(*~
        <docu>
            <summary>
                Clears the message content.
                <remarks>
                    <note type="important">
                        This method is exposed for Rpc calls, for testing purposes. Rpc calls of this method must not be used in production code
                    </note>
                </remarks>
            </summary>
        </docu>
~*)
{attribute 'TcRpcEnable'}
METHOD Clear
_mime.TimeStamp := DT#1970-01-01-00:00;
_mime.Text := '';
_mime.Identity := 0;
_mime.Category := eMessageCategory.All;
_mime.Cycle := 0;
_mime.PerCycleCount := 0;
_mime.Pinned := FALSE;
END_METHOD

METHOD PROTECTED Compose : TcoMessage
VAR_INPUT
    Text : STRING(TcoMessengerEnv.MAX_MESSAGE_TEXT_LENGHT);
    Category : eMessageCategory;
END_VAR
IF (_Parent <> 0 AND_THEN _Parent.Context <> 0 AND_THEN _Parent.Context.RealTimeClock <> 0) THEN
    Compose.TimeStamp := _Parent.Context.RealTimeClock.NowLocal();
    Compose.Text := Text;
    Compose.Identity := _Parent.Identity;
    Compose.Category := Category;
    Compose.Cycle := _Parent.Context.StartCycleCount;
    Compose.MessageDigest := Digest(Text, THIS^._Parent.Context.Environment.Messaging.MessageDigestMethod);
END_IF;
END_METHOD

(*~
        <docu>
            <summary>
                Adds message of 'critical' category to the message queue.
                Use this category when a critical error occured, that is not recoverable by the means of software (reset/restore) and a detailed inspection is required.
            </summary>
        </docu>
~*)
METHOD PUBLIC Critical : ITcoMessageProperties
VAR_INPUT
    (*~
        <docu>
            <summary>
                Arbitrary message string.
            </summary>
        </docu>
    ~*)
    Message : STRING(TcoMessengerEnv.MAX_MESSAGE_TEXT_LENGHT);
END_VAR
Critical := THIS^.Post(Message, eMessageCategory.Critical);
END_METHOD

(*~
        <docu>
            <summary>
                Adds message of 'debug' category to the message queue.
                Use when you need to report debug information for you as programmer.
            </summary>
        </docu>
~*)
METHOD PUBLIC Debug : ITcoMessageProperties
VAR_INPUT
    (*~
        <docu>
            <summary>
                Arbitrary message string.
            </summary>
        </docu>
    ~*)
    Message : STRING(TcoMessengerEnv.MAX_MESSAGE_TEXT_LENGHT);
END_VAR
Debug := THIS^.Post(Message, eMessageCategory.Debug);
END_METHOD

METHOD Digest : DWORD
VAR_INPUT
    Text : Tc2_System.T_MaxString;
    inDigestType : eMessageDigestMethod;
END_VAR
CASE inDigestType OF
    eMessageDigestMethod.CRC8:
        Digest := TcoCRC_8(Text);
    eMessageDigestMethod.CRC16:
        Digest := TcoCRC_16(Text);
    eMessageDigestMethod.CRC32:
        Digest := TcoCRC_32(Text);
ELSE
    Digest := 0;
END_CASE
END_METHOD

(*~
        <docu>
            <summary>
                Adds message of 'error' category to the message queue.
                Use this categoty when there is a failure that cannot be immediately recovered and an intervention is needed. This is typically a situation when a device fails
                to deliver expected result.
                Do not use this category to report information about failed process like measurement or detection.
            </summary>
        </docu>
~*)
METHOD PUBLIC Error : ITcoMessageProperties
VAR_INPUT
    (*~
        <docu>
            <summary>
                Arbitrary message string.
            </summary>
        </docu>
    ~*)
    Message : STRING(TcoMessengerEnv.MAX_MESSAGE_TEXT_LENGHT);
END_VAR
Error := THIS^.Post(Message, eMessageCategory.Error);
END_METHOD

{attribute 'hide'}
METHOD FB_init : BOOL
VAR_INPUT
    bInitRetains : BOOL; // if TRUE, the retain variables are initialized (warm start / cold start)
    bInCopyCode : BOOL; // if TRUE, the instance afterwards gets moved into the copy code (online change)
    ParentObject : ITcoObject;
END_VAR
_Parent := ParentObject;
_contextIdentity := ParentObject.Identity;
END_METHOD

(*~
        <docu>
            <summary>
                Adds message of 'information' category to the message queue.
                Use when you want to deliver information to the user, that has only informative character and does not adversely affect a process.
            </summary>
        </docu>
~*)
METHOD PUBLIC Info : ITcoMessageProperties
VAR_INPUT
    (*~
        <docu>
            <summary>
                Arbitrary message string.
            </summary>
        </docu>
    ~*)
    Message : STRING(TcoMessengerEnv.MAX_MESSAGE_TEXT_LENGHT);
END_VAR
Info := THIS^.Post(Message, eMessageCategory.Info);
END_METHOD

METHOD PRIVATE LogMessage
VAR_IN_OUT
    inMessage : TcoMessage;
END_VAR
VAR
    _index : INT;
    _freeIndex : INT;
END_VAR
CASE _Parent.Context.Environment.Messaging.MessengerLoggingMethod OF
    eMessengerLogMethod.OnEventRisen:
        IF (_Parent.Context.Environment.Messaging.MessageDigestMethod = eMessageDigestMethod.NONE) THEN
            inMessage.MessageDigest := Digest(inMessage.Text, eMessageDigestMethod.CRC32);
        END_IF

        _freeIndex := 0;

        FOR _index := 0 TO MDS_MAX_INDEX DO
            IF (_mds[_index].Cycle = inMessage.Cycle - 1 OR _mds[_index].Cycle = inMessage.Cycle) AND_THEN
                (_mds[_index].Digest = inMessage.MessageDigest) AND_THEN
                (_mds[_index].Category = inMessage.Category) THEN
                _mds[_index].Cycle := inMessage.Cycle;
                RETURN;
            END_IF

            IF ((_mds[_index].Cycle <> inMessage.Cycle - 1) AND (_mds[_index].Cycle <> inMessage.Cycle)) THEN
                _freeIndex := _index;
            END_IF
        END_FOR

        IF (_freeIndex <= THIS^.MDS_MAX_INDEX) THEN
            _mds[_freeIndex].Digest := inMessage.MessageDigest;
            _mds[_freeIndex].Cycle := inMessage.Cycle;
            _mds[_freeIndex].Category := inMessage.Category;
            _Parent.Context.Logger.PushMessage(inMessage);
        END_IF;
    eMessengerLogMethod.Continuous:
        _Parent.Context.Logger.PushMessage(inMessage);
END_CASE
END_METHOD

(*~
        <docu>
            <summary>
                Adds message of 'notification' category to the message queue.
                Use this category when you want to report a notification that may be of interest to the user, but does not adveresly affect a process.
            </summary>
        </docu>
~*)
METHOD Notify : ITcoMessageProperties
VAR_INPUT
    (*~
        <docu>
            <summary>
                Arbitrary message string.
            </summary>
        </docu>
    ~*)
    Message : STRING(TcoMessengerEnv.MAX_MESSAGE_TEXT_LENGHT);
END_VAR
Notify := THIS^.Post(Message, eMessageCategory.Notification);
END_METHOD

METHOD OnCondition : ITcoMessages
VAR_INPUT
    inCondition : BOOL;
END_VAR
IF (inCondition) THEN
    _condition := eMessageCondition.Active;
ELSE
    _condition := eMessageCondition.Inactive;
END_IF

OnCondition := THIS^;
END_METHOD

(*~
    <docu>
        <summary>
            Pins this message that no other message will override it.
            The messenger won't accept new messages until acknowledged in diagnostics view by user, unipenned by `Unpin()` methods or cleared by `Clear()` method
            of this messenger.
        </summary>
        <note type="important">
            Pinned messages do no accept incomming messages on the same messenger. The incomming messages will be though the context logger when active.
        </note>
    </docu>
~*)
//~
{attribute 'hide'}
{attribute 'obsolete' := 'This method must be called exclusively over ITcoMessageProperties interface'}
//~
METHOD Pin : ITcoMessageProperties
IF (_Parent <> 0 AND_THEN _Parent.Context <> 0) THEN
    IF (_pinnable AND_THEN _mime.Cycle = _Parent.Context.StartCycleCount) THEN
        _mime.Pinned := TRUE;
    END_IF;
END_IF;

Pin := THIS^;
END_METHOD

(*~
    <docu>
        <summary>
            Gets `true` when this messanger is pinned (awaiting acknowledgement in diagnostics view).
        </summary>
    </docu>
~*)
PROPERTY Pinned : BOOL
GET
Pinned := _mime.Pinned AND_THEN tmpMessageText = _mime.Text;
END_GET
END_PROPERTY

(*~
        <docu>
            <summary>
                Creates message of given category for this messenger.
            </summary>
        </docu>
~*)
METHOD PUBLIC Post : ITcoMessageProperties
VAR_INPUT
    (*~
        <docu>
            <summary>
                Arbitrary message string.
            </summary>
        </docu>
    ~*)
    Message : STRING(TcoMessengerEnv.MAX_MESSAGE_TEXT_LENGHT);
    (*~
        <docu>
            <summary>
                Message category.
            </summary>
        </docu>
    ~*)
    Category : eMessageCategory;
END_VAR
VAR
    _wouldBeMime : TcoMessage;
END_VAR
Post := THIS^;
tmpMessageText := Message;
_pinnable := FALSE;

IF (_condition = eMessageCondition.Inactive) THEN
    _condition := eMessageCondition.Unconditional;
    RETURN;
END_IF

_condition := eMessageCondition.Unconditional;

IF (_Parent <> 0 AND_THEN _Parent.Context <> 0 AND_THEN _Parent.Context.Environment <> 0 AND_THEN _Parent.Context.Environment.Messaging <> 0) THEN
    IF (Category < THIS^._Parent.Context.Environment.Messaging.MinLevel OR _Parent.Context.Environment.Messaging.IsSuspended) THEN
        RETURN;
    END_IF;

    IF (NOT _mime.Pinned) THEN
        _mime.PerCycleCount := _mime.PerCycleCount + 1;
        _wouldBeMime := Compose(Message, Category);
        _wouldBeMime.PerCycleCount := _mime.PerCycleCount;
    ELSIF (_mime.Pinned AND_THEN (_mime.Text <> Message OR _mime.Category <> Category)) THEN
        IF (_mime.PerCycleCount < 255) THEN
            _mime.PerCycleCount := _mime.PerCycleCount + 1;
        END_IF;
    END_IF;

    // Same cycle filter for most important messge.
    IF (_mime.Cycle = _Parent.Context.StartCycleCount) THEN
        IF (_wouldBeMime.Category > _mime.Category) AND (NOT _mime.Pinned) THEN
            _mime := _wouldBeMime;
        END_IF;
    ELSE
        // Different cycle
        IF (NOT _mime.Pinned) THEN
            _wouldBeMime.PerCycleCount := 1;
            _mime := _wouldBeMime;
        END_IF;
    END_IF;

    _pinnable := TRUE;
    LogMessage(_wouldBeMime);
END_IF;
END_METHOD

(*~
        <docu>
            <summary>
                Adds message of 'programming error' category to the message queue.
                Use this category to inform about a possible programming error, defect in settings or missing information at a level of programming or system or process settings.
            </summary>
        </docu>
~*)
METHOD PUBLIC Programming : ITcoMessageProperties
VAR_INPUT
    (*~
        <docu>
            <summary>
                Arbitrary message string.
            </summary>
        </docu>
    ~*)
    Message : STRING(TcoMessengerEnv.MAX_MESSAGE_TEXT_LENGHT);
END_VAR
Programming := THIS^.Post(Message, eMessageCategory.ProgrammingError);
END_METHOD

PROPERTY StringBuilder : REFERENCE TO StringBuilder
GET
VAR
END_VAR
VAR_INST
    _lastCycleAccess : ULINT;
END_VAR
IF (__ISVALIDREF(refStringBuilder)) THEN
    StringBuilder REF= refStringBuilder;
ELSE
    StringBuilder REF= _conflictingStringBuilder;
END_IF
END_GET
END_PROPERTY

(*~
        <docu>
            <summary>
                Adds message of 'trace' category to the message queue.
                Use when you need to track detailed information about internal states of the program for detailed visibility.
                This is lowest level of category that can be used in production, for detailed observation of PLC program.
            </summary>
        </docu>
~*)
METHOD PUBLIC Trace : ITcoMessageProperties
VAR_INPUT
    (*~
        <docu>
            <summary>
                Arbitrary message string.
            </summary>
        </docu>
    ~*)
    Message : STRING(TcoMessengerEnv.MAX_MESSAGE_TEXT_LENGHT);
END_VAR
Trace := THIS^.Post(Message, eMessageCategory.Trace);
END_METHOD

(*~
    <docu>
        <summary>
            Unpins this messenger.
        </summary>
    </docu>
~*)
METHOD UnPin
IF (_mime.Pinned) THEN
    IF (_Parent <> 0 AND_THEN _Parent.Context <> 0) THEN
        THIS^.Post('Message unpinned by the controller.', eMessageCategory.Info);
    END_IF;
END_IF;

_mime.Pinned := FALSE;
END_METHOD

(*~
        <docu>
            <summary>
                Adds message of 'warning' category to the message queue.
                Use this category when you want to report to the user an information about a possible problem, that may adversly affect a process.
                Information in this cateogory aims to help the user to identify a problem, the cause of such problem does not necessarily stops the process.
            </summary>
        </docu>
~*)
METHOD PUBLIC Warning : ITcoMessageProperties
VAR_INPUT
    (*~
        <docu>
            <summary>
                Arbitrary message string.
            </summary>
        </docu>
    ~*)
    Message : STRING(TcoMessengerEnv.MAX_MESSAGE_TEXT_LENGHT);
END_VAR
Warning := THIS^.Post(Message, eMessageCategory.Warning);
END_METHOD

END_FUNCTION_BLOCK

// ---- POUs/Utilities/TcoCRC_8.TcPOU
FUNCTION INTERNAL TcoCRC_8 : BYTE
VAR_INPUT
    In : Tc2_System.T_MaxString;
END_VAR
VAR
    crc : BYTE := 16#FF;
    pDataArr : POINTER TO BYTE;
    pByte : POINTER TO BYTE;
    bByte : BYTE;
    i : INT;
    maxIndex : INT;
END_VAR
VAR_STAT CONSTANT
    //Precalculated values for polynomial generator of value 0x1D
    CRC_TABLE : ARRAY[0..255] OF BYTE := [
        16#00,
        16#1D,
        16#3A,
        16#27,
        16#74,
        16#69,
        16#4E,
        16#53,
        16#E8,
        16#F5,
        16#D2,
        16#CF,
        16#9C,
        16#81,
        16#A6,
        16#BB,
        16#CD,
        16#D0,
        16#F7,
        16#EA,
        16#B9,
        16#A4,
        16#83,
        16#9E,
        16#25,
        16#38,
        16#1F,
        16#02,
        16#51,
        16#4C,
        16#6B,
        16#76,
        16#87,
        16#9A,
        16#BD,
        16#A0,
        16#F3,
        16#EE,
        16#C9,
        16#D4,
        16#6F,
        16#72,
        16#55,
        16#48,
        16#1B,
        16#06,
        16#21,
        16#3C,
        16#4A,
        16#57,
        16#70,
        16#6D,
        16#3E,
        16#23,
        16#04,
        16#19,
        16#A2,
        16#BF,
        16#98,
        16#85,
        16#D6,
        16#CB,
        16#EC,
        16#F1,
        16#13,
        16#0E,
        16#29,
        16#34,
        16#67,
        16#7A,
        16#5D,
        16#40,
        16#FB,
        16#E6,
        16#C1,
        16#DC,
        16#8F,
        16#92,
        16#B5,
        16#A8,
        16#DE,
        16#C3,
        16#E4,
        16#F9,
        16#AA,
        16#B7,
        16#90,
        16#8D,
        16#36,
        16#2B,
        16#0C,
        16#11,
        16#42,
        16#5F,
        16#78,
        16#65,
        16#94,
        16#89,
        16#AE,
        16#B3,
        16#E0,
        16#FD,
        16#DA,
        16#C7,
        16#7C,
        16#61,
        16#46,
        16#5B,
        16#08,
        16#15,
        16#32,
        16#2F,
        16#59,
        16#44,
        16#63,
        16#7E,
        16#2D,
        16#30,
        16#17,
        16#0A,
        16#B1,
        16#AC,
        16#8B,
        16#96,
        16#C5,
        16#D8,
        16#FF,
        16#E2,
        16#26,
        16#3B,
        16#1C,
        16#01,
        16#52,
        16#4F,
        16#68,
        16#75,
        16#CE,
        16#D3,
        16#F4,
        16#E9,
        16#BA,
        16#A7,
        16#80,
        16#9D,
        16#EB,
        16#F6,
        16#D1,
        16#CC,
        16#9F,
        16#82,
        16#A5,
        16#B8,
        16#03,
        16#1E,
        16#39,
        16#24,
        16#77,
        16#6A,
        16#4D,
        16#50,
        16#A1,
        16#BC,
        16#9B,
        16#86,
        16#D5,
        16#C8,
        16#EF,
        16#F2,
        16#49,
        16#54,
        16#73,
        16#6E,
        16#3D,
        16#20,
        16#07,
        16#1A,
        16#6C,
        16#71,
        16#56,
        16#4B,
        16#18,
        16#05,
        16#22,
        16#3F,
        16#84,
        16#99,
        16#BE,
        16#A3,
        16#F0,
        16#ED,
        16#CA,
        16#D7,
        16#35,
        16#28,
        16#0F,
        16#12,
        16#41,
        16#5C,
        16#7B,
        16#66,
        16#DD,
        16#C0,
        16#E7,
        16#FA,
        16#A9,
        16#B4,
        16#93,
        16#8E,
        16#F8,
        16#E5,
        16#C2,
        16#DF,
        16#8C,
        16#91,
        16#B6,
        16#AB,
        16#10,
        16#0D,
        16#2A,
        16#37,
        16#64,
        16#79,
        16#5E,
        16#43,
        16#B2,
        16#AF,
        16#88,
        16#95,
        16#C6,
        16#DB,
        16#FC,
        16#E1,
        16#5A,
        16#47,
        16#60,
        16#7D,
        16#2E,
        16#33,
        16#14,
        16#09,
        16#7F,
        16#62,
        16#45,
        16#58,
        16#0B,
        16#16,
        16#31,
        16#2C,
        16#97,
        16#8A,
        16#AD,
        16#B0,
        16#E3,
        16#FE,
        16#D9,
        16#C4];
END_VAR

TcoCRC_8 := crc;
pDataArr := ADR(In);
maxIndex := Tc2_Standard.LEN(In) - 1;

IF (pDataArr = 0) OR (maxIndex < 0) THEN
    RETURN;
END_IF

FOR i := 0 TO maxIndex BY 1 DO
    pByte := pDataArr + INT_TO_UINT(i);
    bByte := pByte^;
    crc := CRC_TABLE[bByte XOR crc];
END_FOR

TcoCRC_8 := crc;

END_FUNCTION

// ---- POUs/Utilities/TcoCRC_16.TcPOU
FUNCTION INTERNAL TcoCRC_16 : WORD
VAR_INPUT
    In : Tc2_System.T_MaxString;
END_VAR
VAR
    crc : WORD := 16#FFFF;
    pDataArr : POINTER TO BYTE;
    pByte : POINTER TO BYTE;
    bByte : BYTE;
    i : INT;
    maxIndex : INT;
END_VAR
VAR_STAT CONSTANT
    //Precalculated values for polynomial generator of value 0x1021
    CRC_TABLE : ARRAY[0..255] OF WORD := [
        16#0000,
        16#1021,
        16#2042,
        16#3063,
        16#4084,
        16#50A5,
        16#60C6,
        16#70E7,
        16#8108,
        16#9129,
        16#A14A,
        16#B16B,
        16#C18C,
        16#D1AD,
        16#E1CE,
        16#F1EF,
        16#1231,
        16#0210,
        16#3273,
        16#2252,
        16#52B5,
        16#4294,
        16#72F7,
        16#62D6,
        16#9339,
        16#8318,
        16#B37B,
        16#A35A,
        16#D3BD,
        16#C39C,
        16#F3FF,
        16#E3DE,
        16#2462,
        16#3443,
        16#0420,
        16#1401,
        16#64E6,
        16#74C7,
        16#44A4,
        16#5485,
        16#A56A,
        16#B54B,
        16#8528,
        16#9509,
        16#E5EE,
        16#F5CF,
        16#C5AC,
        16#D58D,
        16#3653,
        16#2672,
        16#1611,
        16#0630,
        16#76D7,
        16#66F6,
        16#5695,
        16#46B4,
        16#B75B,
        16#A77A,
        16#9719,
        16#8738,
        16#F7DF,
        16#E7FE,
        16#D79D,
        16#C7BC,
        16#48C4,
        16#58E5,
        16#6886,
        16#78A7,
        16#0840,
        16#1861,
        16#2802,
        16#3823,
        16#C9CC,
        16#D9ED,
        16#E98E,
        16#F9AF,
        16#8948,
        16#9969,
        16#A90A,
        16#B92B,
        16#5AF5,
        16#4AD4,
        16#7AB7,
        16#6A96,
        16#1A71,
        16#0A50,
        16#3A33,
        16#2A12,
        16#DBFD,
        16#CBDC,
        16#FBBF,
        16#EB9E,
        16#9B79,
        16#8B58,
        16#BB3B,
        16#AB1A,
        16#6CA6,
        16#7C87,
        16#4CE4,
        16#5CC5,
        16#2C22,
        16#3C03,
        16#0C60,
        16#1C41,
        16#EDAE,
        16#FD8F,
        16#CDEC,
        16#DDCD,
        16#AD2A,
        16#BD0B,
        16#8D68,
        16#9D49,
        16#7E97,
        16#6EB6,
        16#5ED5,
        16#4EF4,
        16#3E13,
        16#2E32,
        16#1E51,
        16#0E70,
        16#FF9F,
        16#EFBE,
        16#DFDD,
        16#CFFC,
        16#BF1B,
        16#AF3A,
        16#9F59,
        16#8F78,
        16#9188,
        16#81A9,
        16#B1CA,
        16#A1EB,
        16#D10C,
        16#C12D,
        16#F14E,
        16#E16F,
        16#1080,
        16#00A1,
        16#30C2,
        16#20E3,
        16#5004,
        16#4025,
        16#7046,
        16#6067,
        16#83B9,
        16#9398,
        16#A3FB,
        16#B3DA,
        16#C33D,
        16#D31C,
        16#E37F,
        16#F35E,
        16#02B1,
        16#1290,
        16#22F3,
        16#32D2,
        16#4235,
        16#5214,
        16#6277,
        16#7256,
        16#B5EA,
        16#A5CB,
        16#95A8,
        16#8589,
        16#F56E,
        16#E54F,
        16#D52C,
        16#C50D,
        16#34E2,
        16#24C3,
        16#14A0,
        16#0481,
        16#7466,
        16#6447,
        16#5424,
        16#4405,
        16#A7DB,
        16#B7FA,
        16#8799,
        16#97B8,
        16#E75F,
        16#F77E,
        16#C71D,
        16#D73C,
        16#26D3,
        16#36F2,
        16#0691,
        16#16B0,
        16#6657,
        16#7676,
        16#4615,
        16#5634,
        16#D94C,
        16#C96D,
        16#F90E,
        16#E92F,
        16#99C8,
        16#89E9,
        16#B98A,
        16#A9AB,
        16#5844,
        16#4865,
        16#7806,
        16#6827,
        16#18C0,
        16#08E1,
        16#3882,
        16#28A3,
        16#CB7D,
        16#DB5C,
        16#EB3F,
        16#FB1E,
        16#8BF9,
        16#9BD8,
        16#ABBB,
        16#BB9A,
        16#4A75,
        16#5A54,
        16#6A37,
        16#7A16,
        16#0AF1,
        16#1AD0,
        16#2AB3,
        16#3A92,
        16#FD2E,
        16#ED0F,
        16#DD6C,
        16#CD4D,
        16#BDAA,
        16#AD8B,
        16#9DE8,
        16#8DC9,
        16#7C26,
        16#6C07,
        16#5C64,
        16#4C45,
        16#3CA2,
        16#2C83,
        16#1CE0,
        16#0CC1,
        16#EF1F,
        16#FF3E,
        16#CF5D,
        16#DF7C,
        16#AF9B,
        16#BFBA,
        16#8FD9,
        16#9FF8,
        16#6E17,
        16#7E36,
        16#4E55,
        16#5E74,
        16#2E93,
        16#3EB2,
        16#0ED1,
        16#1EF0];
END_VAR

TcoCRC_16 := crc;
pDataArr := ADR(In);
maxIndex := Tc2_Standard.LEN(In) - 1;

IF (pDataArr = 0) OR (maxIndex < 0) THEN
    RETURN;
END_IF

FOR i := 0 TO maxIndex BY 1 DO
    pByte := pDataArr + INT_TO_UINT(i);
    bByte := pByte^;
    crc := SHL(crc, 8) XOR CRC_TABLE[SHR(crc, 8) XOR bByte];
END_FOR

TcoCRC_16 := crc;

END_FUNCTION

// ---- POUs/Utilities/TcoCRC_32.TcPOU
FUNCTION INTERNAL TcoCRC_32 : DWORD
VAR_INPUT
    In : Tc2_System.T_MaxString;
END_VAR
VAR
    crc : DWORD := 16#FFFFFFFF;
    pDataArr : POINTER TO BYTE;
    pByte : POINTER TO BYTE;
    bByte : BYTE;
    i : INT;
    maxIndex : INT;
    posD : UDINT;
    pos : BYTE;
END_VAR
VAR_STAT CONSTANT
    //Precalculated values for polynomial generator of value 0x04C11DB7
    CRC_TABLE : ARRAY[0..255] OF DWORD := [
        16#00000000,
        16#04C11DB7,
        16#09823B6E,
        16#0D4326D9,
        16#130476DC,
        16#17C56B6B,
        16#1A864DB2,
        16#1E475005,
        16#2608EDB8,
        16#22C9F00F,
        16#2F8AD6D6,
        16#2B4BCB61,
        16#350C9B64,
        16#31CD86D3,
        16#3C8EA00A,
        16#384FBDBD,
        16#4C11DB70,
        16#48D0C6C7,
        16#4593E01E,
        16#4152FDA9,
        16#5F15ADAC,
        16#5BD4B01B,
        16#569796C2,
        16#52568B75,
        16#6A1936C8,
        16#6ED82B7F,
        16#639B0DA6,
        16#675A1011,
        16#791D4014,
        16#7DDC5DA3,
        16#709F7B7A,
        16#745E66CD,
        16#9823B6E0,
        16#9CE2AB57,
        16#91A18D8E,
        16#95609039,
        16#8B27C03C,
        16#8FE6DD8B,
        16#82A5FB52,
        16#8664E6E5,
        16#BE2B5B58,
        16#BAEA46EF,
        16#B7A96036,
        16#B3687D81,
        16#AD2F2D84,
        16#A9EE3033,
        16#A4AD16EA,
        16#A06C0B5D,
        16#D4326D90,
        16#D0F37027,
        16#DDB056FE,
        16#D9714B49,
        16#C7361B4C,
        16#C3F706FB,
        16#CEB42022,
        16#CA753D95,
        16#F23A8028,
        16#F6FB9D9F,
        16#FBB8BB46,
        16#FF79A6F1,
        16#E13EF6F4,
        16#E5FFEB43,
        16#E8BCCD9A,
        16#EC7DD02D,
        16#34867077,
        16#30476DC0,
        16#3D044B19,
        16#39C556AE,
        16#278206AB,
        16#23431B1C,
        16#2E003DC5,
        16#2AC12072,
        16#128E9DCF,
        16#164F8078,
        16#1B0CA6A1,
        16#1FCDBB16,
        16#018AEB13,
        16#054BF6A4,
        16#0808D07D,
        16#0CC9CDCA,
        16#7897AB07,
        16#7C56B6B0,
        16#71159069,
        16#75D48DDE,
        16#6B93DDDB,
        16#6F52C06C,
        16#6211E6B5,
        16#66D0FB02,
        16#5E9F46BF,
        16#5A5E5B08,
        16#571D7DD1,
        16#53DC6066,
        16#4D9B3063,
        16#495A2DD4,
        16#44190B0D,
        16#40D816BA,
        16#ACA5C697,
        16#A864DB20,
        16#A527FDF9,
        16#A1E6E04E,
        16#BFA1B04B,
        16#BB60ADFC,
        16#B6238B25,
        16#B2E29692,
        16#8AAD2B2F,
        16#8E6C3698,
        16#832F1041,
        16#87EE0DF6,
        16#99A95DF3,
        16#9D684044,
        16#902B669D,
        16#94EA7B2A,
        16#E0B41DE7,
        16#E4750050,
        16#E9362689,
        16#EDF73B3E,
        16#F3B06B3B,
        16#F771768C,
        16#FA325055,
        16#FEF34DE2,
        16#C6BCF05F,
        16#C27DEDE8,
        16#CF3ECB31,
        16#CBFFD686,
        16#D5B88683,
        16#D1799B34,
        16#DC3ABDED,
        16#D8FBA05A,
        16#690CE0EE,
        16#6DCDFD59,
        16#608EDB80,
        16#644FC637,
        16#7A089632,
        16#7EC98B85,
        16#738AAD5C,
        16#774BB0EB,
        16#4F040D56,
        16#4BC510E1,
        16#46863638,
        16#42472B8F,
        16#5C007B8A,
        16#58C1663D,
        16#558240E4,
        16#51435D53,
        16#251D3B9E,
        16#21DC2629,
        16#2C9F00F0,
        16#285E1D47,
        16#36194D42,
        16#32D850F5,
        16#3F9B762C,
        16#3B5A6B9B,
        16#0315D626,
        16#07D4CB91,
        16#0A97ED48,
        16#0E56F0FF,
        16#1011A0FA,
        16#14D0BD4D,
        16#19939B94,
        16#1D528623,
        16#F12F560E,
        16#F5EE4BB9,
        16#F8AD6D60,
        16#FC6C70D7,
        16#E22B20D2,
        16#E6EA3D65,
        16#EBA91BBC,
        16#EF68060B,
        16#D727BBB6,
        16#D3E6A601,
        16#DEA580D8,
        16#DA649D6F,
        16#C423CD6A,
        16#C0E2D0DD,
        16#CDA1F604,
        16#C960EBB3,
        16#BD3E8D7E,
        16#B9FF90C9,
        16#B4BCB610,
        16#B07DABA7,
        16#AE3AFBA2,
        16#AAFBE615,
        16#A7B8C0CC,
        16#A379DD7B,
        16#9B3660C6,
        16#9FF77D71,
        16#92B45BA8,
        16#9675461F,
        16#8832161A,
        16#8CF30BAD,
        16#81B02D74,
        16#857130C3,
        16#5D8A9099,
        16#594B8D2E,
        16#5408ABF7,
        16#50C9B640,
        16#4E8EE645,
        16#4A4FFBF2,
        16#470CDD2B,
        16#43CDC09C,
        16#7B827D21,
        16#7F436096,
        16#7200464F,
        16#76C15BF8,
        16#68860BFD,
        16#6C47164A,
        16#61043093,
        16#65C52D24,
        16#119B4BE9,
        16#155A565E,
        16#18197087,
        16#1CD86D30,
        16#029F3D35,
        16#065E2082,
        16#0B1D065B,
        16#0FDC1BEC,
        16#3793A651,
        16#3352BBE6,
        16#3E119D3F,
        16#3AD08088,
        16#2497D08D,
        16#2056CD3A,
        16#2D15EBE3,
        16#29D4F654,
        16#C5A92679,
        16#C1683BCE,
        16#CC2B1D17,
        16#C8EA00A0,
        16#D6AD50A5,
        16#D26C4D12,
        16#DF2F6BCB,
        16#DBEE767C,
        16#E3A1CBC1,
        16#E760D676,
        16#EA23F0AF,
        16#EEE2ED18,
        16#F0A5BD1D,
        16#F464A0AA,
        16#F9278673,
        16#FDE69BC4,
        16#89B8FD09,
        16#8D79E0BE,
        16#803AC667,
        16#84FBDBD0,
        16#9ABC8BD5,
        16#9E7D9662,
        16#933EB0BB,
        16#97FFAD0C,
        16#AFB010B1,
        16#AB710D06,
        16#A6322BDF,
        16#A2F33668,
        16#BCB4666D,
        16#B8757BDA,
        16#B5365D03,
        16#B1F740B4];
END_VAR

TcoCRC_32 := crc;
pDataArr := ADR(In);
maxIndex := Tc2_Standard.LEN(In) - 1;

IF (pDataArr = 0) OR (maxIndex < 0) THEN
    RETURN;
END_IF

FOR i := 0 TO maxIndex BY 1 DO
    pByte := pDataArr + INT_TO_UINT(i);
    bByte := pByte^;
    posD := SHR(crc, 24) XOR bByte;
    pos := UDINT_TO_BYTE(posD);
    crc := SHL(crc, 8) XOR CRC_TABLE[pos];
END_FOR

TcoCRC_32 := crc;

END_FUNCTION

// ---- POUs/Compatibility/TcoContextNfCompatibility.TcPOU
FUNCTION_BLOCK FINAL TcoContextNfCompatibility EXTENDS TcoContextCompatibility

METHOD PROTECTED FINAL Main
END_METHOD

METHOD PUBLIC VolatileClose
THIS^._Close();
END_METHOD

METHOD PUBLIC VolatileOpen
THIS^._Open();
END_METHOD

END_FUNCTION_BLOCK

// ---- POUs/ImplicitChecks/CheckBounds.TcPOU
// Implicitly generated code : DO NOT EDIT
FUNCTION CheckBounds : DINT
VAR_INPUT
    index, lower, upper : DINT;
END_VAR
// User defined local variables
VAR
    sMessageLow : STRING := 'CheckBounds: Index too low (%d)';
    sMessageHigh : STRING := 'CheckBounds: Index too high (%d)';
END_VAR

// Implicitly generated code : Only an Implementation suggestion
{noflow}
IF index < lower THEN
    CheckBounds := lower;
    ADSLOGDINT(msgCtrlMask := ADSLOG_MSGTYPE_ERROR, msgFmtStr := sMessageLow, dintArg := index);
ELSIF index > upper THEN
    CheckBounds := upper;
    ADSLOGDINT(msgCtrlMask := ADSLOG_MSGTYPE_ERROR, msgFmtStr := sMessageHigh, dintArg := index);
ELSE
    CheckBounds := index;
END_IF

{flow}

END_FUNCTION

// ---- POUs/ImplicitChecks/CheckDivDInt.TcPOU
// Implicitly generated code : DO NOT EDIT
FUNCTION CheckDivDInt : DINT
VAR_INPUT
    divisor : DINT;
END_VAR

// Implicitly generated code : Only an Implementation suggestion
{noflow}
IF divisor = 0 THEN
    CheckDivDInt := 1;
ELSE
    CheckDivDInt := divisor;
END_IF;
{flow}

END_FUNCTION

// ---- POUs/ImplicitChecks/CheckDivLInt.TcPOU
// Implicitly generated code : DO NOT EDIT
FUNCTION CheckDivLInt : LINT
VAR_INPUT
    divisor : LINT;
END_VAR

// Implicitly generated code : Only an Implementation suggestion
{noflow}
IF divisor = 0 THEN
    CheckDivLInt := 1;
ELSE
    CheckDivLInt := divisor;
END_IF;
{flow}

END_FUNCTION

// ---- POUs/ImplicitChecks/CheckDivLReal.TcPOU
// Implicitly generated code : DO NOT EDIT
FUNCTION CheckDivLReal : LREAL
VAR_INPUT
    divisor : LREAL;
END_VAR

// Implicitly generated code : Only an Implementation suggestion
{noflow}
IF divisor = 0 THEN
    CheckDivLReal := 1;
ELSE
    CheckDivLReal := divisor;
END_IF;
{flow}

END_FUNCTION

// ---- POUs/ImplicitChecks/CheckDivReal.TcPOU
// Implicitly generated code : DO NOT EDIT
FUNCTION CheckDivReal : REAL
VAR_INPUT
    divisor : REAL;
END_VAR

// Implicitly generated code : Only an Implementation suggestion
{noflow}
IF divisor = 0 THEN
    CheckDivReal := 1;
ELSE
    CheckDivReal := divisor;
END_IF;
{flow}

END_FUNCTION

// ---- POUs/ImplicitChecks/CheckLRangeSigned.TcPOU
// Implicitly generated code : DO NOT EDIT
FUNCTION CheckLRangeSigned : LINT
VAR_INPUT
    value, lower, upper : LINT;
END_VAR

// Implicitly generated code : Only an Implementation suggestion
{noflow}
IF (value < lower) THEN
    CheckLRangeSigned := lower;
ELSIF (value > upper) THEN
    CheckLRangeSigned := upper;
ELSE
    CheckLRangeSigned := value;
END_IF

{flow}

END_FUNCTION

// ---- POUs/ImplicitChecks/CheckLRangeUnsigned.TcPOU
// Implicitly generated code : DO NOT EDIT
FUNCTION CheckLRangeUnsigned : ULINT
VAR_INPUT
    value, lower, upper : ULINT;
END_VAR

// Implicitly generated code : Only an Implementation suggestion
{noflow}
IF (value < lower) THEN
    CheckLRangeUnsigned := lower;
ELSIF (value > upper) THEN
    CheckLRangeUnsigned := upper;
ELSE
    CheckLRangeUnsigned := value;
END_IF

{flow}

END_FUNCTION

// ---- POUs/ImplicitChecks/CheckPointer.TcPOU
// Implicitly generated code : DO NOT EDIT
FUNCTION CheckPointer : POINTER TO BYTE
VAR_INPUT
    ptToTest : POINTER TO BYTE; // Destination address of the pointer
    iSize : DINT; // Size of the type the pointer points to. (e.g: 20 for POINTER TO ARRAY [0..9] OF INT)
    iGran : DINT; // Granularity of the pointer access. This is the size of the biggest non-structured data type in the type the pointer points to. (e.g: 2 for POINTER TO ARRAY [0..9] OF INT)
    bWrite : BOOL; // Indicates read or write Access. TRUE = write access.
END_VAR

// Implicitly generated code : Only an Implementation suggestion
{noflow}
IF ptToTest = 0 THEN
    ADSLOGSTR(ADSLOG_MSGTYPE_ERROR OR ADSLOG_MSGTYPE_STRING, 'CheckPointer failed due to invalid address.', '');
ELSIF iSize <= 0 THEN
    ADSLOGSTR(ADSLOG_MSGTYPE_ERROR OR ADSLOG_MSGTYPE_STRING, 'CheckPointer failed due to invalid size.', '');
ELSIF iGran <= 0 THEN
    ADSLOGSTR(ADSLOG_MSGTYPE_ERROR OR ADSLOG_MSGTYPE_STRING, 'CheckPointer failed due to invalid granularity.', '');
    // -> Please note that the following memory area check is time consuming:
    //ELSIF F_CheckMemoryArea(pData:=ptToTest,nSize:=DINT_TO_UDINT(iSize)) = E_TcMemoryArea.Unknown THEN
//    ADSLOGSTR(ADSLOG_MSGTYPE_ERROR OR ADSLOG_MSGTYPE_STRING,'CheckPointer failed due to unknown memory area.','');
END_IF

CheckPointer := ptToTest;
{flow}

END_FUNCTION

// ---- POUs/ImplicitChecks/CheckRangeSigned.TcPOU
// Implicitly generated code : DO NOT EDIT
FUNCTION CheckRangeSigned : DINT
VAR_INPUT
    value, lower, upper : DINT;
END_VAR

// Implicitly generated code : Only an Implementation suggestion
{noflow}
IF (value < lower) THEN
    CheckRangeSigned := lower;
ELSIF (value > upper) THEN
    CheckRangeSigned := upper;
ELSE
    CheckRangeSigned := value;
END_IF

{flow}

END_FUNCTION

// ---- POUs/ImplicitChecks/CheckRangeUnsigned.TcPOU
// Implicitly generated code : DO NOT EDIT
FUNCTION CheckRangeUnsigned : UDINT
VAR_INPUT
    value, lower, upper : UDINT;
END_VAR

// Implicitly generated code : Only an Implementation suggestion
{noflow}
IF (value < lower) THEN
    CheckRangeUnsigned := lower;
ELSIF (value > upper) THEN
    CheckRangeUnsigned := upper;
ELSE
    CheckRangeUnsigned := value;
END_IF

{flow}

END_FUNCTION

// ---- POUs/Prototypes/TcoComponent/TcoComponent.TcPOU
(*~
    <docu>
        <summary>
            Basic class for components.
        </summary>
    </docu>
~*)
FUNCTION_BLOCK ABSTRACT TcoComponent EXTENDS TcoObject IMPLEMENTS ITcoComponent
VAR
    {attribute 'hide'}
    _serviceContexCycle : ULINT;
    (*~
    <docu>
        <summary>
            True if component is in service mode.
        </summary>
    </docu>
~*)
    {attribute clr [RenderIgnore()]}
    _inServiceMode : BOOL;
END_VAR

CheckIfIsInServiceMode();

METHOD INTERNAL CheckIfIsInServiceMode
VAR
    _myContextCycleCount : ULINT;
END_VAR
_myContextCycleCount := Context.StartCycleCount;
//When component.Service() is called "before" invoking its task _serviceContexCycle is equal to Context.StartCycleCount
//When component.Service() is called "after" invoking its task (_serviceContexCycle + 1) is equal to Context.StartCycleCount
//otherwise _serviceContexCycle should be lower then Context.StartCycleCount until Context.StartCycleCount overflow its range
//which should occur cca every 585 mil years at 1ms PLC task.
_inServiceMode := _serviceContexCycle = _myContextCycleCount OR (_serviceContexCycle + 1) = _myContextCycleCount;
END_METHOD

(*~
    <docu>
        <summary>
            Gets whether the component is in serviceable state. Serviceable state is when `Service` method is called cyclicaly.
        </summary>
    </docu>
~*)
PROPERTY IsService : BOOL
GET
CheckIfIsInServiceMode();
IsService := _inServiceMode;
END_GET
END_PROPERTY

(*~
    <docu>
        <summary>
            Restores this instance to the Ready state. Can be called explicitly or from within one of the restore mechanisms.
        </summary>
    </docu>
~*)
METHOD ABSTRACT Restore : ITcoRestorable
END_METHOD

(*~
    <docu>
        <summary>
            Executes the logic for manual-maintenance control.
        </summary>
    </docu>
~*)
METHOD PUBLIC FINAL Service
_serviceContexCycle := Context.StartCycleCount;
ServiceMode();
END_METHOD

(*~
    <docu>
        <summary>
            Custom service (manual, maintenance) logic.
            This method must be implemented in derived class.
        </summary>
    </docu>
~*)
METHOD PROTECTED ABSTRACT ServiceMode
END_METHOD

END_FUNCTION_BLOCK

// ---- POUs/Prototypes/TcoComponent/TcoSignalInfo.TcPOU
(*~
    <docu>
        <summary>
            Provides symbol information about a I/O signal.
            <note type="important">
                 `SymbolPath` can only contain string of 255 characters.
            </note>
            <note type="tip">
                 This block is partially extended by IVF to provide more information about the symbol.
            </note>
        </summary>
    </docu>
~*)
FUNCTION_BLOCK TcoSignalInfo
VAR
    (*~
    <docu>
        <summary>
            Symbol path of the Signal.
            <note type="important">
                 SymbolPath can only contain string of 255 characters.
            </note>
        </summary>
    </docu>
    ~*)
    SymbolPath : STRING[255];
    {attribute 'hide'}
    pLast : POINTER TO ULINT;
END_VAR

(*~
    <docu>
        <summary>
            Gets symbol path of the variable that is associated to hardware I/O.
        </summary>
    </docu>
~*)
METHOD PUBLIC GetSignalInfo
VAR_INPUT
    (*~
    <docu>
        <summary>
            Size of the variable. Is typicaly determined by `SIZEOF` opreator: SIZEOF(Variable)
        </summary>
    </docu>
    ~*)
    ioSIZE : UDINT;
    (*~
    <docu>
        <summary>
            Pointer to the variable is typically determined by `ADR` operator ADR(Variable)
        </summary>
    </docu>
    ~*)
    pVARIABLE : POINTER TO ULINT;
END_VAR
VAR_STAT
    {attribute 'hide'}
    json : Tc3_JsonXml.FB_JsonReadWriteDatatype;
END_VAR
IF (pLast <> pVARIABLE) THEN
    SymbolPath := json.GetSymbolNameByAddress(nData := ioSIZE, pData := pVARIABLE);
    pLast := pVARIABLE;
END_IF;
END_METHOD

END_FUNCTION_BLOCK

// ---- POUs/Prototypes/TcoDialog/TcoCustomizedDialog/TcoCustomizedDialog.TcPOU
(*~
    <docu>
        <summary>
            Provides customized dialog to interact with the user.
         </summary>
        <example>
            [!code-pas[StandardDialog](~/../TcOpen/src/TcoInspectors/src/XAE/XAE/TcoInspectorsTests/POUs/Examples/ExampleContext.TcPOU?name=StandardDialog)]
            [!code-csharp[DialogInitialization](~/../TcOpen/src/TcoInspectors/tests/Sandbox.TcoInspectors.Wpf/App.xaml.cs?name=DialogProxyServiceInitialization)]
        </example>
    </docu>
~*)
FUNCTION_BLOCK TcoCustomizedDialog EXTENDS TcoDialogBase IMPLEMENTS ITcoCustomizedDialogFormat, ITcoCustomizedDialogAnswer
VAR
    _text : STRING(500);
    _caption : STRING(255);
    _hasOption1 : BOOL;
    _hasOption2 : BOOL;
    _hasOption3 : BOOL;
    _hasOption4 : BOOL;
    _contentOption1 : STRING;
    _contentOption2 : STRING;
    _contentOption3 : STRING;
    _contentOption4 : STRING;
    _answer : eCustomizedDialogAnswer;
    _dialogType : eDialogType;
    _rTrig : R_TRIG;
    _imageSource : STRING(255);
    _imageHeight : REAL;
    _imageWidth : REAL;
END_VAR

SUPER^();

{attribute 'hide'}
{attribute 'obsolete' := 'You should access the property via `ITcoDialogAnswer)` interface.'}
(*~
    <docu>
        <summary>
            Gets the answer from the dialog.
         </summary>
    </docu>
~*)
PROPERTY Answer : eCustomizedDialogAnswer
GET
Answer := _answer;
END_GET
END_PROPERTY

METHOD INTERNAL ClearInfos
VAR_INPUT
END_VAR
_imageSource := '';
_caption := '';
_text := '';
_dialogType := eDialogType.Undefined;
END_METHOD

METHOD PROTECTED OnStart
SUPER^.OnStart();
_answer := eCustomizedDialogAnswer.Invoked;
END_METHOD

METHOD Restore : ITcoRestorable
VAR_INPUT
END_VAR
SUPER^.Restore();
ClearInfos();
_answer := eCustomizedDialogAnswer.NoAnswer;
END_METHOD

(*~
    <docu>
        <summary>
            Shows the customized dialog.
            <note type="important">
                In order for the dialog to be displayed to the user user application must initialized in the user application.
                How to set up the observer in a WPF see `TcOpen.Inxton.TcoCore.Wpf.DialogProxyService`.
            </note>
         </summary>
    </docu>
~*)
METHOD Show : ITcoCustomizedDialogFormat
THIS^.Invoke();
SUPER^();
_hasOption1 := FALSE;
_hasOption2 := FALSE;
_hasOption3 := FALSE;
_hasOption4 := FALSE;
_contentOption1 := '';
_contentOption2 := '';
_contentOption3 := '';
_contentOption4 := '';
ClearInfos();
Show := THIS^;

IF THIS^._taskState = eTaskState.Done AND _answer <> eCustomizedDialogAnswer.Invoked AND _answer <> eCustomizedDialogAnswer.NoAnswer THEN
    SUPER^.Restore();
    THIS^.ClearInfos();
END_IF;
END_METHOD

(*~
    <docu>
        <summary>
            Shows the dialog , closig this dialog is possibe  by external signal such as HW button press. Only one answer exclusively in same time is evaluated
            <note type="important">
                In order for the dialog to be displayed to the user user application must initialized in the user application.
                How to set up the observer in a WPF see `TcOpen.Inxton.TcoCore.Wpf.DialogProxyService`.
            </note>
         </summary>
    </docu>
~*)
METHOD ShowWithExternalClose : ITcoCustomizedDialogFormat
VAR_INPUT
    (*~
    <docu>
        <summary>
            If True dialog is closed , and answer result is `eCustomizedDialogAnswer.Option1`
        </summary>
    </docu>
    ~*)
    inOption1AnswerSignal : BOOL := FALSE;
    (*~
    <docu>
        <summary>
            If True dialog is closed , and answer result is `eCustomizedDialogAnswer.Option2`
        </summary>
    </docu>
    ~*)
    inOption2AnswerSignal : BOOL := FALSE;
    (*~
    <docu>
        <summary>
            If True dialog is closed , and answer result is `eCustomizedDialogAnswer.Option3`
        </summary>
    </docu>
    ~*)
    inOption3AnswerSignal : BOOL := FALSE;
    (*~
    <docu>
        <summary>
            If True dialog is closed , and answer result is `eCustomizedDialogAnswer.Option4`
        </summary>
    </docu>
    ~*)
    inOption4AnswerSignal : BOOL := FALSE;
END_VAR
THIS^.Invoke();
SUPER^();
_hasOption1 := FALSE;
_hasOption2 := FALSE;
_hasOption3 := FALSE;
_hasOption4 := FALSE;
_contentOption1 := '';
_contentOption2 := '';
_contentOption3 := '';
_contentOption4 := '';
ClearInfos();
ShowWithExternalClose := THIS^;
_rTrig(CLK := inOption1AnswerSignal XOR inOption2AnswerSignal XOR inOption3AnswerSignal XOR inOption4AnswerSignal);

IF _rTrig.q THEN
    IF inOption1AnswerSignal THEN
        ;
        _answer := eCustomizedDialogAnswer.Option1;
    ELSIF inOption2AnswerSignal THEN
        ;
        _answer := eCustomizedDialogAnswer.Option2;
    ELSIF inOption3AnswerSignal THEN
        ;
        _answer := eCustomizedDialogAnswer.Option3;
    ELSIF inOption4AnswerSignal THEN
        ;
        _answer := eCustomizedDialogAnswer.Option4;
    END_IF;
END_IF

IF THIS^._taskState = eTaskState.Done AND _answer <> eDialogAnswer.Invoked THEN
    SUPER^.Restore();
    THIS^.ClearInfos();
END_IF;
END_METHOD

(*~
    <docu>
        <summary>
            Sets the caption of the dialog window.
         </summary>
    </docu>
~*)
{attribute 'hide'}
{attribute 'obsolete' := 'You should access the method via `Show()` method.'}
METHOD WithCaption : ITcoCustomizedDialogAnswer
VAR_INPUT
    inCaption : STRING(255);
END_VAR
_caption := inCaption;
WithCaption := THIS^;
END_METHOD

(*~
    <docu>
        <summary>
            Sets the image source of the dialog window.
         </summary>
    </docu>
~*)
{attribute 'hide'}
{attribute 'obsolete' := 'You should access the method via `Show()` method.'}
METHOD WithImage : ITcoCustomizedDialogAnswer
VAR_INPUT
    inSource : STRING(255);
    inHeight : REAL;
    inWidth : REAL;
END_VAR
_imageSource := inSource;
_imageHeight := inHeight;
_imageWidth := inWidth;
WithImage := THIS^;
END_METHOD

(*~
    <docu>
        <summary>
            Sets that the `Visibility` and `Content`  of button (Option1).This button should be available in the dialog prompt.
         </summary>
    </docu>
~*)
{attribute 'hide'}
{attribute 'obsolete' := 'You should access the method via `Show()` method.'}
METHOD WithOption1 : ITcoCustomizedDialogAnswer
VAR_INPUT
    inContent : STRING;
END_VAR
_hasOption1 := TRUE;
_contentOption1 := inContent;
WithOption1 := THIS^;
END_METHOD

(*~
    <docu>
        <summary>
            Sets that the `Visibility` and `Content`  of button (Option2).This button should be available in the dialog prompt.
         </summary>
    </docu>
~*)
{attribute 'hide'}
{attribute 'obsolete' := 'You should access the method via `Show()` method.'}
METHOD WithOption2 : ITcoCustomizedDialogAnswer
VAR_INPUT
    inContent : STRING;
END_VAR
_hasOption2 := TRUE;
_contentOption2 := inContent;
WithOption2 := THIS^;
END_METHOD

(*~
    <docu>
        <summary>
            Sets that the `Visibility` and `Content`  of button (Option3).This button should be available in the dialog prompt.
         </summary>
    </docu>
~*)
{attribute 'hide'}
{attribute 'obsolete' := 'You should access the method via `Show()` method.'}
METHOD WithOption3 : ITcoCustomizedDialogAnswer
VAR_INPUT
    inContent : STRING;
END_VAR
_hasOption3 := TRUE;
_contentOption3 := inContent;
WithOption3 := THIS^;
END_METHOD

(*~
    <docu>
        <summary>
            Sets that the `Visibility` and `Content`  of button (Option4).This button should be available in the dialog prompt.
         </summary>
    </docu>
~*)
{attribute 'hide'}
{attribute 'obsolete' := 'You should access the method via `Show()` method.'}
METHOD WithOption4 : ITcoCustomizedDialogAnswer
VAR_INPUT
    inContent : STRING;
END_VAR
_hasOption4 := TRUE;
_contentOption4 := inContent;
WithOption4 := THIS^;
END_METHOD

(*~
    <docu>
        <summary>
            Sets the text of the dialog window.
         </summary>
    </docu>
~*)
{attribute 'hide'}
{attribute 'obsolete' := 'You should access the method via `Show()` method.'}
METHOD WithText : ITcoCustomizedDialogAnswer
VAR_INPUT
    inText : STRING(500);
END_VAR
_text := inText;
WithText := THIS^;
END_METHOD

METHOD WithType : ITcoCustomizedDialogAnswer
VAR_INPUT
    inDialogType : eDialogType;
END_VAR
_dialogType := inDialogType;
WithType := THIS^;
END_METHOD

END_FUNCTION_BLOCK

// ---- POUs/Prototypes/TcoDialog/TcoDialogBase.TcPOU
(*~
    <docu>
        <summary>
            Base block for interactive dialogs.
         </summary>
    </docu>
~*)
FUNCTION_BLOCK ABSTRACT TcoDialogBase EXTENDS TcoRemoteTask

SUPER^();

{attribute 'hide'}
METHOD PUBLIC FB_init : BOOL
VAR_INPUT
    bInitRetains : BOOL; // if TRUE, the retain variables are initialized (warm start / cold start)
    bInCopyCode : BOOL; // if TRUE, the instance afterwards gets moved into the copy code (online change)
    ParentObject : ITcoObject;
END_VAR
END_METHOD

METHOD PROTECTED OnStart
SUPER^.OnStart();
END_METHOD

END_FUNCTION_BLOCK

// ---- POUs/Prototypes/TcoRemoteTask/TcoRemoteTask.TcPOU
(*~
    <docu>
        <summary>
            Remote tasks delegates its execution to C#.
            When this task is invoked a C# method will be called. To initiliaze <code>RemoteTask</code> with C# method use the <code>Initiliaze</code> or <code>InitializeExclusively</code> method.
            <code>
                    partial void PexConstructor(IVortexObject parent, string readableTail, string symbolTail)
                    {
                        _remoteTaskInstance.InitializeExclusively(Create);
                        //_remoteTaskInstance.Initialize(Create);
                    }

                    private bool Create()
                    {
                        //your code.
                        return true;
                    }
            </code>
        </summary>
        <remarks>Inxton is required for this feature to work</remarks>
    </docu>
~*)
FUNCTION_BLOCK TcoRemoteTask EXTENDS TcoTask
VAR
    {attribute clr [RenderIgnore()]}
    _isInitialized : BOOL;
    {attribute clr [RenderIgnore()]}
    _hasException : BOOL;
    {attribute clr [RenderIgnore()]}
    _startSignature : STRING;
    {attribute clr [RenderIgnore()]}
    _doneSignarure : STRING;
    {attribute clr [RenderIgnore()]}
    _exceptionMessage : STRING(255);
END_VAR

IF Execute() THEN
    //IF (_invokeRequest) THEN
    IF (NOT THIS^._isInitialized) THEN
        Messenger.Programming('Remote call not initialized.');
    END_IF;

    //END_IF
    IF (THIS^._hasException OR THIS^._exceptionMessage <> '') THEN
        _startSignature := '';
        ThrowWhen(TRUE);
    END_IF;

    DoneWhen(_startSignature <> '' AND_THEN _startSignature = _doneSignarure);
END_IF

IF (THIS^._hasException) THEN
    Messenger.Error(THIS^._exceptionMessage);
END_IF;

{attribute 'hide'}
METHOD PUBLIC FB_init : BOOL
VAR_INPUT
    bInitRetains : BOOL; // if TRUE, the retain variables are initialized (warm start / cold start)
    bInCopyCode : BOOL; // if TRUE, the instance afterwards gets moved into the copy code (online change)
    ParentObject : ITcoObject;
END_VAR
END_METHOD

METHOD PROTECTED OnStart
_startSignature := ULINT_TO_STRING(THIS^.Context.RealTimeClock.TickClock());
_doneSignarure := '';
_hasException := FALSE;
_exceptionMessage := '';
END_METHOD

(*~
    <docu>
        <summary>
            Restores this instance to the Ready state. Can be called explicitly or from within one of the restore mechanisms.
            <para>
                See also <see cref="PlcDocu.TcoCore.TcoTask.AutoRestorable()"/>
            </para>
        </summary>
    </docu>
~*)
METHOD Restore : ITcoRestorable
_startSignature := '';
_doneSignarure := '';
_hasException := FALSE;
_exceptionMessage := '';
Restore := SUPER^.Restore();
END_METHOD

END_FUNCTION_BLOCK

// ---- POUs/Prototypes/TcoTask/TcoTask.TcPOU
(*~
    <docu>
        <summary>
            Provides basic task execution. Task is started by calling the <see cref="PlcDocu.TcoCore.TcoTask.Invoke()"/> method.
            The  <see cref="PlcDocu.TcoCore.TcoTask.Execute()"/> method returns true, until the task is `Done`.
            <para>
                To get the actual state of the task,
                <see cref="PlcDocu.TcoCore.TcoTask.Ready"/>,
                <see cref="PlcDocu.TcoCore.TcoTask.Busy"/>,
                <see cref="PlcDocu.TcoCore.TcoTask.Error"/>
                and <see cref="PlcDocu.TcoCore.TcoTask.Done"/> properties are available.
            </para>
        </summary>
        <example>
            Declaration part of the 'TcoTask' example.
        </example>
        <example>
            [!code-pas[Main](~/../TcOpen/src/TcoApplicationExamples/XaeAppExamples/PlcAppExamples/POUs/Task/AskForTheFavor_Task.TcPOU?name=TaskExampleDeclarations)]
        </example>
        <example>
            Implementation part of the 'TcoTask' example.
        </example>
        <example>
            [!code-pas[Main](~/../TcOpen/src/TcoApplicationExamples/XaeAppExamples/PlcAppExamples/POUs/Task/AskForTheFavor_Task.TcPOU?name=TaskBodyExampleCode)]
        </example>
        <example>
            Example of the invoking this example 'TcoTask' instance 'outside' of the instance and wait if it ends-up in 'DONE' state or in 'ERROR' state.
        </example>
        <example>
            [!code-pas[Main](~/../TcOpen/src/TcoApplicationExamples/XaeAppExamples/PlcAppExamples/POUs/Sequencer/MakeAnOfferThatCantBeRefused.TcPOU?name=TaskExternalUseExample)]
        </example>
    </docu>
~*)
FUNCTION_BLOCK TcoTask EXTENDS TcoObject IMPLEMENTS ITcoTask, ITcoTaskStatus
VAR
    {attribute clr [ReadOnly()]}
    _taskState : eTaskState;
    {attribute 'hide'}
    _nextExpectedCycle : ULINT;
    {attribute 'hide'}
    _AutoRestorable : BOOL;
    {attribute 'hide'}
    _StartCycleCount : ULINT;
    {attribute 'hide'}
    _MyParentsChangeStateCycle : ULINT;
    {attribute 'hide'}
    _MyParentsLastChangeState : INT;
    {attribute 'hide'}
    _exectuteCallCycle : ULINT;
    (*~
    <docu>
        <summary>
            Use to restore this instance to the Ready state. The value is than set to FALSE.
        </summary>
    </docu>
~*)
    {attribute addProperty Name "<#Restore request#>"}
    _restoreRequest : BOOL;
    (*~
    <docu>
        <summary>
            Use to start the execution of the task from Ready state or from Done state by performing the rising edge.
            <p>Analogously to the xExecute signal of the <a href="https://plcopen.org/sites/default/files/downloads/creating_plcopen_compliant_function_block_libraries.pdf" title="Title"> PLCopen </a> motion function blocks.</p>
        </summary>
    </docu>
~*)
    {attribute addProperty Name "<#Invoke request#>"}
    _invokeRequest : BOOL;
    (*~
    <docu>
        <summary>
            Use to abort the executing task and set this instance back to the Ready state.
            The value is than set to FALSE.
        </summary>
    </docu>
~*)
    {attribute addProperty Name "<#Abort request#>"}
    _abortRequest : BOOL;
    (*~
    <docu>
        <summary>
            Use to determine if the task execution is enabled for example from the HMI application.
            This value is read only, to modify it use the property <see cref="PlcDocu.TcoCore.TcoTask.Enabled()"/>
        </summary>
    </docu>
~*)
    {attribute addProperty Name "<#Enabled#>"}
    {attribute clr [ReadOnly()]}
    _enabled : BOOL := TRUE;
    (*~
    <docu>
        <summary>
            Indicates whether the task is in serviceable state. The default state 'serviceable' that means that the task
            can be invoked from the higher-level application. The serviceable state is cancelled when the immediate parent is `ITcoServiceable`
            and at the same time the parent is not in servicebable state. `TcoComponent` is serviceable, in order for the component's task to be
            invokable from higher-level application component must call `Service` method to induce the component into serviceable state.
        </summary>
    </docu>
    ~*)
    {attribute addProperty Name "<#Serviceable#>"}
    {attribute clr [ReadOnly()]}
    {attribute clr [RenderIgnore()]}
    _isServiceable : BOOL;
END_VAR
VAR
    {attribute 'hide'}
    _executionTimer : Tc2_Standard.TON;
    {attribute clr [ReadOnly()]}
    _elapsedTime : TIME;
END_VAR

(*~
    <docu>
        <summary>
            Aborts the execution of this task and restores the ready state.
        </summary>
    </docu>
~*)
METHOD Abort
IF THIS^._taskState = eTaskState.Busy THEN
    THIS^.Messenger.Trace('<#Task aborted.#>');
    OnAbort();
    THIS^.Restore();
END_IF
END_METHOD

(*~
    <docu>
        <summary>
            Gets whether this instance is auto restorable. This is depends on the parent's settings; the value of this property is given by the parent of this object.
            This value is assigned after download by calling the implicit method <c>FB_init()</c> of the parent object and cannot be changed during runtime.
            The <c>AutoRestorable</c> property of this objects is retrieved from the <c>EnableAutoRestore</c> property of the parent object.
            This is done by calling the <c>CheckIfAutoRestoreEnabledByParent()</c> method inside the implicit method <c>FB_init()</c> after download.
            If this instance is the auto restorable it will call the <see cref="PlcDocu.TcoCore.TcoTask.Restore()"/> method if:
            <para>
                1.) The <see cref="PlcDocu.TcoCore.TcoTask.Invoke()"/> method has not been called for one or more cycles and starts to be called again.
            </para>
            <para>
                2.)	Parent object of this instance changes its state.
            </para>
            <para>
                See also <see cref="PlcDocu.TcoCore.TcoTask.EnableAutoRestore()"/>
            </para>
        </summary>
    </docu>
~*)
PROPERTY AutoRestorable : BOOL
GET
AutoRestorable := _AutoRestorable;
END_GET
END_PROPERTY

(*~
    <docu>
        <summary>
            Private method called each time that the <see cref="PlcDocu.TcoCore.TcoTask.Execute()"/> method is called. If this instance is auto restorable, this method ensures calling the <see cref="PlcDocu.TcoCore.TcoTask.Restore()"/> method if:
            <para>
                1.)	Parent object of this instance changes its state in this Plc cycle.
            </para>
            <para>
                2.)	Parent object of this instance changes its state no mather when and this instance has not yet process this change.
            </para>
            <para>
                3.) The <see cref="PlcDocu.TcoCore.TcoTask.Invoke()"/> method has not been called for one or more cycles and starts to be called again.
            </para>
            <para>
                See also <see cref="PlcDocu.TcoCore.TcoTask.AutoRestorable()"/>
            </para>
            <para>
                See also <see cref="PlcDocu.TcoCore.TcoTask.EnableAutoRestore()"/>
            </para>
        </summary>
    </docu>
~*)
METHOD PRIVATE AutoRestore
VAR
    _MyParent_TcoState : ITcoState := 0;
    _MyParent_ChangeStateCycle : ULINT;
    _MyParent_LastChangeState : INT;
END_VAR
// If the parent of this instance is TcoState type or its derived type and the parent
// EnableAutoRestore property is set to TRUE, this instance determines the value
// of its own AutoRestorable property by calling CheckIfAutoRestoreEnabledByParent
// after each download.
IF _AutoRestorable THEN
    IF __QUERYINTERFACE(THIS^.Parent, _MyParent_TcoState) THEN
        _MyParent_ChangeStateCycle := _MyParent_TcoState.LastStateChangeCycle;
        _MyParent_LastChangeState := _MyParent_TcoState.State;
    END_IF;

    //If OnStateChange event of the parent has occured, the value of the parent's
    //StartCycleCount property is stored into its ChangeStateCycle property.
    //Each child has to deal with it individually in the next call of its body,
    //restore itself, and copy the parent's ChangeStateCycle property into the
    //child's own property.
    IF _MyParent_ChangeStateCycle <> _MyParentsChangeStateCycle THEN
        Restore();
        _MyParentsChangeStateCycle := _MyParent_ChangeStateCycle;
    END_IF

    IF _MyParent_LastChangeState <> _MyParentsLastChangeState THEN
        Restore();
        _MyParentsLastChangeState := _MyParent_LastChangeState;
    END_IF
END_IF
END_METHOD

(*~
    <docu>
        <summary>
            Gets whether the task is executing.
        </summary>
    </docu>
~*)
{attribute 'monitoring' := 'variable'}
PROPERTY Busy : BOOL
GET
Busy := THIS^._taskState = eTaskState.Busy;
END_GET
END_PROPERTY

(*~
    <docu>
        <summary>
            Gets the context of this object.
            This context is given by declaration, its value is assigned after download by calling the implicit method <c>FB_init()</c> and cannot be changed during runtime.
        </summary>
    </docu>
~*)
PROPERTY Context : ITcoContext
GET
Context := THIS^.Parent.Context;
END_GET
END_PROPERTY

(*~
    <docu>
        <summary>
            Gets whether the task has succesfully completed the  execution and did not enter into the Error state.
        </summary>
    </docu>
~*)
{attribute 'monitoring' := 'variable'}
PROPERTY Done : BOOL
GET
Done := THIS^._taskState = eTaskState.Done;
PrivateDetectExecuteCall();
END_GET
END_PROPERTY

(*~
    <docu>
        <summary>
            Completes the execution of this task when ```inCondition``` is true; the task transitions into ```Done``` state.
        </summary>
    </docu>
~*)
METHOD DoneWhen
VAR_INPUT
    inCondition : BOOL;
END_VAR
IF (inCondition AND THIS^._taskState = eTaskState.Busy) THEN
    THIS^._taskState := eTaskState.Done;
    THIS^.Messenger.Trace('<#Task done.#>');
    OnDone();
END_IF;
END_METHOD

(*~
    <docu>
        <summary>
            Gets the elapsed time of the execution of this task.
            <remarks>
                <note type="important">
                    Uses `TIME` type. It might be not sutable for tasks running longer than 49 days.
                </note>
            </remarks>
        </summary>
    </docu>
~*)
{attribute 'monitoring' := 'variable'}
PROPERTY PUBLIC ElapsedTime : TIME
GET
ElapsedTime := _elapsedTime;
END_GET
END_PROPERTY

(*~
    <docu>
        <summary>
            Gets whether the task execution is enabled.
            The task can start with <see cref="PlcDocu.TcoCore.TcoTask.Invoke()"/> method call only when this property si TRUE.
            If the task is ```Busy``` and this property transitions to ```FALSE```, the task stops execution and enters ```Error``` state.
        </summary>
    </docu>
~*)
{attribute 'monitoring' := 'variable'}
PROPERTY Enabled : BOOL
GET
Enabled := _enabled;
END_GET
SET
_enabled := Enabled;
END_SET
END_PROPERTY

(*~
    <docu>
        <summary>
            Returns true if the task has is in error state. To be able to start the the task again, <see cref="PlcDocu.TcoCore.TcoTask.Restore()"/> method needs to be called before
            restarting it again calling <see cref="PlcDocu.TcoCore.TcoTask.Invoke()"/> method.
        </summary>
    </docu>
~*)
{attribute 'monitoring' := 'variable'}
PROPERTY Error : BOOL
GET
Error := THIS^._taskState = eTaskState.Error;
END_GET
END_PROPERTY

(*~
    <docu>
        <summary>
            Returns true if the task is Busy, otherwise false.
            This method needs to be called cyclically.
        </summary>
    </docu>
~*)
METHOD Execute : BOOL
VAR
    _serviceableParent : ITcoServiceable;
END_VAR
VAR
    tmpTimeDiff : TIME;
END_VAR
// Detects if parent is in serviceable state to enable manual invoke of the task from the HMI/SCADA system.
IF (THIS^.Parent <> 0) THEN
    _isServiceable := TRUE;

    IF (__QUERYINTERFACE(THIS^.Parent, _serviceableParent)) THEN
        IF (NOT _serviceableParent.IsService) THEN
            THIS^._invokeRequest := FALSE;
            _isServiceable := FALSE;
        END_IF
    END_IF
END_IF;

IF (THIS^.Parent.Context <> 0) THEN
    _exectuteCallCycle := THIS^.Parent.Context.StartCycleCount;
END_IF;

//Triggering Invoke from remote system
IF (THIS^._taskState = eTaskState.Ready AND THIS^._invokeRequest) THEN
    THIS^.Invoke();
END_IF;

THIS^._invokeRequest := FALSE;

//Triggering Abort from remote system
IF ((THIS^._taskState = eTaskState.Requested OR THIS^._taskState = eTaskState.Busy) AND THIS^._abortRequest) THEN
    THIS^.Abort();
    THIS^._abortRequest := FALSE;
END_IF;

//Triggering Restore from remote system
IF (THIS^._restoreRequest) THEN
    THIS^.Restore();
    THIS^._restoreRequest := FALSE;
END_IF;

IF NOT _enabled THEN
    IF THIS^._taskState = eTaskState.Requested THEN
        THIS^.Messenger.Post('<#Task cannot start; Enabled property is FALSE.#>', eMessageCategory.Info);
        THIS^.Restore();
    END_IF

    IF THIS^._taskState = eTaskState.Busy THEN
        THIS^.Messenger.Post('<#Running task entered Error state when the Enabled property transitioned to FALSE during task execution.#>',
            eMessageCategory.Error);

        THIS^._taskState := eTaskState.Error;
    END_IF
END_IF;

CheckIfCalledCyclically();
AutoRestore();

IF (THIS^._taskState = eTaskState.Requested) THEN
    _executionTimer(IN := FALSE);
    THIS^._taskState := eTaskState.Busy;
    THIS^.Messenger.Trace('<#Task started.#>');
    THIS^.OnStart();
END_IF;

IF (THIS^._taskState = eTaskState.Error) THEN
    WhileError();
END_IF;

Execute := (THIS^._taskState = eTaskState.Busy);

IF (Execute) THEN
    _executionTimer(IN := Execute, PT := T#49D);
    _elapsedTime := _executionTimer.ET;
END_IF;
END_METHOD

{attribute 'hide'}
METHOD PUBLIC FB_init : BOOL
VAR_INPUT
    bInitRetains : BOOL; // if TRUE, the retain variables are initialized (warm start / cold start)
    bInCopyCode : BOOL; // if TRUE, the instance afterwards gets moved into the copy code (online change)
    ParentObject : ITcoObject;
END_VAR
_ParentObject := ParentObject;
CheckIfAutoRestoreEnabledByParent();
END_METHOD

(*~
    <docu>
        <summary>
            This method ensures reading out the parent's <see cref="PlcDocu.TcoCore.TcoState.EnableAutoRestore()/> property and writing it into the <see cref="PlcDocu.TcoCore.TcoTask.AutoRestorable()"/> of this instance.
            Calling this method is ensured by calling the implicit method <c>FB_init()</c> after download, or after online change.
        </summary>
    </docu>
~*)
{attribute 'call_after_online_change_slot' := '100'}
METHOD PRIVATE CheckIfAutoRestoreEnabledByParent
VAR
    _MyParent_TcoState : ITcoState := 0;
END_VAR
IF __QUERYINTERFACE(THIS^.Parent, _MyParent_TcoState) THEN
    _AutoRestorable := _MyParent_TcoState.IsAutoRestoreEnabled;
END_IF;
END_METHOD

(*~
    <docu>
        <summary>
            Private method called inside the <see cref="PlcDocu.TcoCore.TcoTask.Execute()"/> method checking the cyclicall calling of this method.
            If this instance is auto restorable, this method ensures calling the <see cref="PlcDocu.TcoCore.TcoTask.Restore()"/> method if
            the <see cref="PlcDocu.TcoCore.TcoTask.Execute()"/> method has not been called for one or more cycles and starts to be called again.
            <para>
                See also <see cref="PlcDocu.TcoCore.TcoTask.AutoRestorable()"/>
            </para>
            <para>
                See also <see cref="PlcDocu.TcoCore.TcoTask.EnableAutoRestore()"/>
            </para>
        </summary>
    </docu>
~*)
{attribute clr [ExcludeFromApiDocumentation()]}
METHOD PRIVATE CheckIfCalledCyclically
VAR
    _MyContextStartCycleCount : ULINT;
END_VAR
//If parent of this instance is TcoState type or its derived type and the parent
//EnableAutoRestore property is set to TRUE, this instance determines the value
//of its own AutoRestorable property by calling CheckIfAutoRestoreEnabledByParent
//after each download.
IF _AutoRestorable THEN
    _MyContextStartCycleCount := THIS^.Context.StartCycleCount;

    //If this instance is AutoRestorable, its body has to be called cyclically,
    //otherwise this instance is restored.
    //This mechanism force the user to call this instance properly,
    //in order to don't miss the OnStateChange() event of the parent
    //in case of the body of this instance isn't called.
    IF _MyContextStartCycleCount > _StartCycleCount + 1 THEN
        Restore();
    END_IF

    _StartCycleCount := _MyContextStartCycleCount;
END_IF
END_METHOD

(*~
    <docu>
        <summary>
            Gets identity of this <see cref ="PlcDocu.TcoCore.TcoTask()"/>.
            This value is assigned after download by calling the implicit method <c>FB_init()</c> and cannot be changed during runtime.
            This variable is used in the higher level applications.
        </summary>
    </docu>
~*)
PROPERTY Identity : ULINT
GET
Identity := _Identity;
END_GET
END_PROPERTY

(*~
    <docu>
        <summary>
            Use to start the execution of the task. The starting is possible from Ready state.
            <para>Moreover it is also possible to start the task again from Done state by performing the '''rising edge''' of the calling of the Invoke() method.</para>
            <p>Analogously to the xExecute signal of the <a href="https://plcopen.org/sites/default/files/downloads/creating_plcopen_compliant_function_block_libraries.pdf" title="Title"> PLCopen </a> motion function blocks.</p>
        </summary>
    </docu>
~*)
METHOD Invoke : ITcoTaskStatus
VAR
    _newInvokeCall : BOOL;
END_VAR
_newInvokeCall := THIS^.Parent.Context.StartCycleCount > _nextExpectedCycle;

IF (THIS^._taskState = eTaskState.Ready OR (THIS^._taskState = eTaskState.Done AND _newInvokeCall)) THEN
    IF _enabled THEN
        THIS^._taskState := eTaskState.Requested;
        THIS^.Messenger.Trace('<#Task requested.#>');
    ELSE
        THIS^.Messenger.Post('Tasks is not enabled.', eMessageCategory.Info);
    END_IF
END_IF

_nextExpectedCycle := THIS^.Parent.Context.StartCycleCount + 1;
Invoke := THIS^;
END_METHOD

(*~
    <docu>
        <summary>
            Executes when task is aborted.
        </summary>
    </docu>
~*)
METHOD PROTECTED OnAbort
END_METHOD

(*~
    <docu>
        <summary>
            Executes when task reaches the ```Done``` state .
        </summary>
    </docu>
~*)
METHOD PROTECTED OnDone
END_METHOD

(*~
    <docu>
        <summary>
            Executes when task reaches the ```Error``` state.
            <para>
                Do not confuse with <see cref="PlcDocu.TcoCore.TcoTask.WhileError()"/>, that is called cyclically until '''Error''' state is left.
            </para>
        </summary>
    </docu>
~*)
METHOD PROTECTED OnError
END_METHOD

(*~
    <docu>
        <summary>
            Executes ones when the task starts (at the moment of transition from the ```Requested``` state into the ```Busy``` state).
        </summary>
    </docu>
~*)
METHOD PROTECTED OnStart
END_METHOD

METHOD PRIVATE PrivateDetectExecuteCall
THIS^.Messenger.OnCondition(THIS^.Parent.Context.StartCycleCount > _exectuteCallCycle + 1)
    .Programming('Cyclic execution of the task not called. Make sure you are calling Execute() method cyclically in the call tree of the context.');
END_METHOD

(*~
    <docu>
        <summary>
            Gets whether the task is ready to be started (Tasks start by calling the <see cref="PlcDocu.TcoCore.TcoTask.Invoke()"/> method).
        </summary>
    </docu>
~*)
{attribute 'monitoring' := 'variable'}
PROPERTY Ready : BOOL
GET
Ready := THIS^._taskState = eTaskState.Ready;
END_GET
END_PROPERTY

(*~
    <docu>
        <summary>
            Restores this instance to the Ready state. Can be called explicitly or from within one of the restore mechanisms.
            <para>
                See also <see cref="PlcDocu.TcoCore.TcoTask.AutoRestorable()"/>
            </para>
        </summary>
    </docu>
~*)
METHOD Restore : ITcoRestorable
THIS^._taskState := eTaskState.Ready;
THIS^.Messenger.Trace('<#Task restored.#>');
Restore := THIS^;
END_METHOD

(*~
    <docu>
        <summary>
            Gets the actual state of this instance.
            <para>
                See <see cref="TcoCore.eTaskState"/> for more details.
            </para>
        </summary>
    </docu>
~*)
{attribute 'monitoring' := 'variable'}
PROPERTY State : eTaskState
GET
State := _taskState;
END_GET
END_PROPERTY

(*~
    <docu>
        <summary>
            When called with ```inCondition``` ```TRUE``` causes transition of the task into the ```Error``` state.
        </summary>
    </docu>
~*)
METHOD ThrowWhen
VAR_INPUT
    inCondition : BOOL;
END_VAR
IF (inCondition) THEN
    THIS^._taskState := eTaskState.Error;
    THIS^.Messenger.Trace('<#Task error thrown.#>');
    OnError();
END_IF
END_METHOD

(*~
    <docu>
        <summary>
            Executes until task is in ```Error``` state .
            <para>
                Do not confuse with <see cref="PlcDocu.TcoCore.TcoTask.OnError()"/>, that is called just ones when '''Error''' state is entered.
            </para>
        </summary>
    </docu>
~*)
METHOD PROTECTED WhileError
END_METHOD

END_FUNCTION_BLOCK

// ---- POUs/Prototypes/TcoDialog/TcoDialog.TcPOU
(*~
    <docu>
        <summary>
            Provides standard dialog to interact with the user.
         </summary>
        <example>
            [!code-pas[StandardDialog](~/../TcOpen/src/TcoInspectors/src/XAE/XAE/TcoInspectorsTests/POUs/Examples/ExampleContext.TcPOU?name=StandardDialog)]
            [!code-csharp[DialogInitialization](~/../TcOpen/src/TcoInspectors/tests/Sandbox.TcoInspectors.Wpf/App.xaml.cs?name=DialogProxyServiceInitialization)]
        </example>
    </docu>
~*)
FUNCTION_BLOCK TcoDialog EXTENDS TcoDialogBase IMPLEMENTS ITcoDialogFormat, ITcoDialogAnswer
VAR
    _text : STRING(500);
    _caption : STRING(255);
    _hasOK : BOOL;
    _hasYes : BOOL;
    _hasNo : BOOL;
    _hasCancel : BOOL;
    _answer : eDialogAnswer;
    _dialogType : eDialogType;
    _rTrig : R_TRIG;
    _imageSource : STRING(255);
    _imageHeight : REAL;
    _imageWidth : REAL;
END_VAR

SUPER^();

{attribute 'hide'}
{attribute 'obsolete' := 'You should access the property via `ITcoDialogAnswer)` interface.'}
(*~
    <docu>
        <summary>
            Gets the answer from the dialog.
         </summary>
    </docu>
~*)
PROPERTY Answer : eDialogAnswer
GET
Answer := _answer;
END_GET
END_PROPERTY

METHOD INTERNAL ClearInfos
VAR_INPUT
END_VAR
_imageSource := '';
_caption := '';
_text := '';
_dialogType := eDialogType.Undefined;
END_METHOD

METHOD PROTECTED OnStart
SUPER^.OnStart();
_answer := eDialogAnswer.Invoked;
END_METHOD

METHOD Restore : ITcoRestorable
VAR_INPUT
END_VAR
SUPER^.Restore();
THIS^.ClearInfos();
_answer := eDialogAnswer.NoAnswer;
END_METHOD

(*~
    <docu>
        <summary>
            Shows the dialog.
            <note type="important">
                In order for the dialog to be displayed to the user user application must initialized in the user application.
                How to set up the observer in a WPF see `TcOpen.Inxton.TcoCore.Wpf.DialogProxyService`.
            </note>
         </summary>
    </docu>
~*)
METHOD Show : ITcoDialogFormat
THIS^.Invoke();
SUPER^();
_hasOK := FALSE;
_hasYes := FALSE;
_hasNo := FALSE;
_hasCancel := FALSE;
ClearInfos();
Show := THIS^;

IF THIS^._taskState = eTaskState.Done AND _answer <> eDialogAnswer.Invoked AND _answer <> eDialogAnswer.NoAnswer THEN
    SUPER^.Restore();
    THIS^.ClearInfos();
END_IF;
END_METHOD

(*~
    <docu>
        <summary>
            Shows the dialog , closig this dialog is possibe  by external signal such as HW button press. Only one answer exclusively in same time is evaluated
            <note type="important">
                In order for the dialog to be displayed to the user user application must initialized in the user application.
                How to set up the observer in a WPF see `TcOpen.Inxton.TcoCore.Wpf.DialogProxyService`.
            </note>
         </summary>
    </docu>
~*)
METHOD ShowWithExternalClose : ITcoDialogFormat
VAR_INPUT
    (*~
    <docu>
        <summary>
            If True dialog is closed , and answer result is `eDialogAnsw.Ok`
        </summary>
    </docu>
    ~*)
    inOkAnswerSignal : BOOL := FALSE;
    (*~
    <docu>
        <summary>
            If True dialog is closed , and answer result is `eDialogAnsw.Yes`
        </summary>
    </docu>
    ~*)
    inYesAnswerSignal : BOOL := FALSE;
    (*~
    <docu>
        <summary>
            If True dialog is closed , and answer result is `eDialogAnsw.No`
        </summary>
    </docu>
    ~*)
    inNoAnswerSignal : BOOL := FALSE;
    (*~
    <docu>
        <summary>
            If True dialog is closed , and answer result is `eDialogAnsw.Cancel`
        </summary>
    </docu>
    ~*)
    inCancelAnswerSignal : BOOL := FALSE;
END_VAR
THIS^.Invoke();
SUPER^();
_hasOK := FALSE;
_hasYes := FALSE;
_hasNo := FALSE;
_hasCancel := FALSE;
ClearInfos();
ShowWithExternalClose := THIS^;
_rTrig(CLK := inOkAnswerSignal XOR inYesAnswerSignal XOR inNoAnswerSignal XOR inCancelAnswerSignal);

IF _rTrig.q THEN
    IF inOkAnswerSignal THEN
        ;
        _answer := eDialogAnswer.Ok;
    ELSIF inYesAnswerSignal THEN
        ;
        _answer := eDialogAnswer.Yes;
    ELSIF inNoAnswerSignal THEN
        ;
        _answer := eDialogAnswer.No;
    ELSIF inCancelAnswerSignal THEN
        ;
        _answer := eDialogAnswer.Cancel;
    END_IF;
END_IF

IF THIS^._taskState = eTaskState.Done AND _answer <> eDialogAnswer.Invoked AND _answer <> eDialogAnswer.NoAnswer THEN
    SUPER^.Restore();
    THIS^.ClearInfos();
END_IF;
END_METHOD

(*~
    <docu>
        <summary>
            Sets the caption of the dialog window.
         </summary>
    </docu>
~*)
{attribute 'hide'}
{attribute 'obsolete' := 'You should access the method via `Show()` method.'}
METHOD WithCaption : ITcoDialogAnswer
VAR_INPUT
    inCaption : STRING(255);
END_VAR
_caption := inCaption;
WithCaption := THIS^;
END_METHOD

(*~
    <docu>
        <summary>
            Sets the image source of the dialog window.
         </summary>
    </docu>
~*)
{attribute 'hide'}
{attribute 'obsolete' := 'You should access the method via `Show()` method.'}
METHOD WithImage : ITcoDialogAnswer
VAR_INPUT
    inSource : STRING(255);
    inHeight : REAL;
    inWidth : REAL;
END_VAR
_imageSource := inSource;
_imageHeight := inHeight;
_imageWidth := inWidth;
WithImage := THIS^;
END_METHOD

(*~
    <docu>
        <summary>
            Sets that the `OK` button should be available in the dialog prompt.
         </summary>
    </docu>
~*)
{attribute 'hide'}
{attribute 'obsolete' := 'You should access the method via `Show()` method.'}
METHOD WithOk : ITcoDialogAnswer
VAR_INPUT
END_VAR
_hasOK := TRUE;
WithOk := THIS^;
END_METHOD

(*~
    <docu>
        <summary>
            Sets the text of the dialog window.
         </summary>
    </docu>
~*)
{attribute 'hide'}
{attribute 'obsolete' := 'You should access the method via `Show()` method.'}
METHOD WithText : ITcoDialogAnswer
VAR_INPUT
    inText : STRING(500);
END_VAR
_text := inText;
WithText := THIS^;
END_METHOD

METHOD WithType : ITcoDialogAnswer
VAR_INPUT
    inDialogType : eDialogType;
END_VAR
_dialogType := inDialogType;
WithType := THIS^;
END_METHOD

(*~
    <docu>
        <summary>
            Sets that the `Yes` and `No` buttons should be available in the dialog prompt.
         </summary>
    </docu>
~*)
{attribute 'hide'}
{attribute 'obsolete' := 'You should access the method via `Show()` method.'}
METHOD WithYesNo : ITcoDialogAnswer
VAR_INPUT
END_VAR
_hasYes := TRUE;
_hasNo := TRUE;
WithYesNo := THIS^;
END_METHOD

(*~
    <docu>
        <summary>
            Sets that the `Yes`, `No` and `Cancel` buttons should be available in the dialog prompt.
         </summary>
    </docu>
~*)
{attribute 'hide'}
{attribute 'obsolete' := 'You should access the method via `Show()` method.'}
METHOD WithYesNoCancel : ITcoDialogAnswer
_hasYes := TRUE;
_hasNo := TRUE;
_hasCancel := TRUE;
WithYesNoCancel := THIS^;
END_METHOD

END_FUNCTION_BLOCK

// ---- POUs/Prototypes/TcoNothing/NO.TcPOU
PROGRAM NO
VAR
    Obj : ITcoObject;
    Structure : TcoStruct;
END_VAR

END_PROGRAM

// ---- POUs/Prototypes/TcoDialog/TcoInputDialog/TcoInputDialog.TcPOU
(*~
    <docu>
        <summary>
            Provides standard dialog to interact with the user and provide fields for values input.
         </summary>

    </docu>
~*)
FUNCTION_BLOCK TcoInputDialog EXTENDS TcoDialogBase IMPLEMENTS ITcoInputDialogAnswer, ITcoInputDialogAnswer
VAR
    _text : STRING(500);
    _caption : STRING(255);
    _hasOK : BOOL;
    _hasYes : BOOL;
    _hasNo : BOOL;
    _answer : eInputDialogAnswer;
    _dialogType : eDialogType;
    _rTrig : R_TRIG;
    _imageSource : STRING(255);
    _imageHeight : REAL;
    _imageWidth : REAL;
    {attribute clr [MemberByIdentity()]}
    _content : TcoInputDialogContentContainer(THIS^);
END_VAR

SUPER^();

(*~
    <docu>
        <summary>
            Gets the answer from the input dialog .
         </summary>
    </docu>
~*)
PROPERTY Answer : eInputDialogAnswer
GET
Answer := _answer;
END_GET
END_PROPERTY

METHOD INTERNAL ClearInfos
VAR_INPUT
END_VAR
_imageSource := '';
_caption := '';
_text := '';
_dialogType := eDialogType.Undefined;
END_METHOD

METHOD PROTECTED OnStart
SUPER^.OnStart();
_answer := eDialogAnswer.Invoked;
END_METHOD

METHOD Restore : ITcoRestorable
VAR_INPUT
END_VAR
SUPER^.Restore();
THIS^.ClearInfos();
_answer := eDialogAnswer.NoAnswer;
END_METHOD

(*~
    <docu>
        <summary>
            Shows the dialog.
            <note type="important">
                In order for the dialog to be displayed to the user user application must initialized in the user application.
                How to set up the observer in a WPF see `TcOpen.Inxton.TcoCore.Wpf.DialogProxyService`.
            </note>
         </summary>
    </docu>
~*)
METHOD Show : ITcoInputDialogFormat
VAR_INPUT
    refContent : REFERENCE TO TcoInputDialogContentContainer;
END_VAR
IF NOT __ISVALIDREF(refContent) THEN
    Messenger.Post('<#Invalid reference axis 1#>', eMessageCategory.ProgrammingError);
    RETURN;
END_IF

_content := refContent;
THIS^.Invoke();
SUPER^();
_hasOK := FALSE;
_hasYes := FALSE;
_hasNo := FALSE;
ClearInfos();
Show := THIS^;

IF THIS^._taskState = eTaskState.Done AND _answer <> eDialogAnswer.Invoked AND _answer <> eDialogAnswer.NoAnswer THEN
    SUPER^.Restore();
    THIS^.ClearInfos();
END_IF;
END_METHOD

(*~
    <docu>
        <summary>
            Shows the dialog , closig this dialog is possibe  by external signal such as HW button press. Only one answer exclusively in same time is evaluated
            <note type="important">
                In order for the dialog to be displayed to the user user application must initialized in the user application.
                How to set up the observer in a WPF see `TcOpen.Inxton.TcoCore.Wpf.DialogProxyService`.
            </note>
         </summary>
    </docu>
~*)
METHOD ShowWithExternalClose : ITcoInputDialogFormat
VAR_IN_OUT
    inoContent : TcoInputDialogContentContainer;
END_VAR
VAR_INPUT
    (*~
    <docu>
        <summary>
            If True dialog is closed , and answer result is `eDialogAnsw.Ok`
        </summary>
    </docu>
    ~*)
    inOkAnswerSignal : BOOL := FALSE;
    (*~
    <docu>
        <summary>
            If True dialog is closed , and answer result is `eDialogAnsw.Yes`
        </summary>
    </docu>
    ~*)
    inYesAnswerSignal : BOOL := FALSE;
    (*~
    <docu>
        <summary>
            If True dialog is closed , and answer result is `eDialogAnsw.No`
        </summary>
    </docu>
    ~*)
    inNoAnswerSignal : BOOL := FALSE;
    (*~
    <docu>
        <summary>
            If True dialog is closed , and answer result is `eDialogAnsw.Cancel`
        </summary>
    </docu>
    ~*)
    inCancelAnswerSignal : BOOL := FALSE;
END_VAR
_content := inoContent;
THIS^.Invoke();
SUPER^();
_hasOK := FALSE;
_hasYes := FALSE;
_hasNo := FALSE;
ClearInfos();
ShowWithExternalClose := THIS^;
_rTrig(CLK := inOkAnswerSignal XOR inYesAnswerSignal XOR inNoAnswerSignal XOR inCancelAnswerSignal);

IF _rTrig.q THEN
    IF inOkAnswerSignal THEN
        ;
        _answer := eDialogAnswer.Ok;
    ELSIF inYesAnswerSignal THEN
        ;
        _answer := eDialogAnswer.Yes;
    ELSIF inNoAnswerSignal THEN
        ;
        _answer := eDialogAnswer.No;
    ELSIF inCancelAnswerSignal THEN
        ;
        _answer := eDialogAnswer.Cancel;
    END_IF;
END_IF

IF THIS^._taskState = eTaskState.Done AND _answer <> eDialogAnswer.Invoked AND _answer <> eDialogAnswer.NoAnswer THEN
    inoContent := _content;
    SUPER^.Restore();
    THIS^.ClearInfos();
END_IF;
END_METHOD

(*~
    <docu>
        <summary>
            Sets the caption of the dialog window.
         </summary>
    </docu>
~*)
{attribute 'hide'}
{attribute 'obsolete' := 'You should access the method via `Show()` method.'}
METHOD WithCaption : ITcoInputDialogAnswer
VAR_INPUT
    inCaption : STRING(255);
END_VAR
_caption := inCaption;
WithCaption := THIS^;
END_METHOD

(*~
    <docu>
        <summary>
            Sets the image source of the dialog window.
         </summary>
    </docu>
~*)
{attribute 'hide'}
{attribute 'obsolete' := 'You should access the method via `Show()` method.'}
METHOD WithImage : ITcoInputDialogAnswer
VAR_INPUT
    inSource : STRING(255);
    inHeight : REAL;
    inWidth : REAL;
END_VAR
_imageSource := inSource;
_imageHeight := inHeight;
_imageWidth := inWidth;
WithImage := THIS^;
END_METHOD

(*~
    <docu>
        <summary>
            Sets that the `OK` button should be available in the dialog prompt.
         </summary>
    </docu>
~*)
{attribute 'hide'}
{attribute 'obsolete' := 'You should access the method via `Show()` method.'}
METHOD WithOk : ITcoInputDialogAnswer
VAR_INPUT
END_VAR
_hasOK := TRUE;
WithOk := THIS^;
END_METHOD

(*~
    <docu>
        <summary>
            Sets the text of the dialog window.
         </summary>
    </docu>
~*)
{attribute 'hide'}
{attribute 'obsolete' := 'You should access the method via `Show()` method.'}
METHOD WithText : ITcoInputDialogAnswer
VAR_INPUT
    inText : STRING(500);
END_VAR
_text := inText;
WithText := THIS^;
END_METHOD

METHOD WithType : ITcoInputDialogAnswer
VAR_INPUT
    inDialogType : eDialogType;
END_VAR
_dialogType := inDialogType;
WithType := THIS^;
END_METHOD

(*~
    <docu>
        <summary>
            Sets that the `Yes` and `No` buttons should be available in the dialog prompt.
         </summary>
    </docu>
~*)
{attribute 'hide'}
{attribute 'obsolete' := 'You should access the method via `Show()` method.'}
METHOD WithYesNo : ITcoInputDialogAnswer
VAR_INPUT
END_VAR
_hasYes := TRUE;
_hasNo := TRUE;
WithYesNo := THIS^;
END_METHOD

END_FUNCTION_BLOCK

// ---- POUs/Prototypes/TcoDialog/TcoInputDialog/TcoInputDialogContentContainer.TcPOU
FUNCTION_BLOCK TcoInputDialogContentContainer EXTENDS TcoObject

END_FUNCTION_BLOCK

// ---- POUs/Prototypes/TcoMomentaryTask/TcoMomentaryTask.TcPOU
(*~
    <docu>
        <summary>
            Provides basic momentary on function.
            <para>
                To get the actual state of the momentary task, <see cref="PlcDocu.TcoCore.TcoMomentaryTask.IsOn()"/>, <see cref="PlcDocu.TcoCore.TcoMomentaryTask.IsOff()"/> and <see cref="PlcDocu.TcoCore.TcoMomentaryTask.State()"/> properties are available.
            </para>
        </summary>
    </docu>
~*)
{attribute addProperty StateOnDesc "<#On#>"}
{attribute addProperty StateOffDesc "<#Off#>"}
FUNCTION_BLOCK TcoMomentaryTask EXTENDS TcoObject IMPLEMENTS ITcoMomentaryTask
VAR
    {attribute clr [ReadOnly()]}
    _state : BOOL;
    (*~
    <docu>
        <summary>
            Use to set the state to the '''TRUE''' value.
        </summary>
    </docu>
~*)
    {attribute addProperty Name "<#Set on request#>"}
    _setOnRequest : BOOL;
    (*~
    <docu>
        <summary>
            Use to determine if the manipulation is enabled for example from the HMI application.
            This value is read only, to modify it use the property <see cref="PlcDocu.TcoCore.TcoMomentaryTask.Enabled()"/>
        </summary>
    </docu>
~*)
    {attribute addProperty Name "<#Enabled#>"}
    {attribute clr [ReadOnly()]}
    _enabled : BOOL := TRUE;
    {attribute 'hide'}
    _StartCycleCount : ULINT;
    (*~
    <docu>
        <summary>
            Indicated whether the task is in serviceable state. The default state 'serviceable' that means that the task
            can be invoked from the higher-level application. The serviceable state is cancelled when the immediate parent is `ITcoServiceable`
            and at the same time the parent is not in servicebable state. `TcoComponent` is serviceable, in order for the component's task to be
            invokable from higher-level application component must call `Service` method to induce the component into serviceable state.
        </summary>
    </docu>
    ~*)
    {attribute addProperty Name "<#Serviceable#>"}
    {attribute clr [ReadOnly()]}
    {attribute clr [RenderIgnore()]}
    _isServiceable : BOOL;
END_VAR

(*~
    <docu>
        <summary>
            Gets the context of this object.
            This context is given by declaration, its value is assigned after download by calling the implicit method <c>FB_init()</c> and cannot be changed during runtime.
        </summary>
    </docu>
~*)
PROPERTY Context : ITcoContext
GET
Context := THIS^.Parent.Context;
END_GET
END_PROPERTY

(*~
    <docu>
        <summary>
            Gets whether the any manipulation with this instance is enabled.
            The change state could be triggered with <see cref="PlcDocu.TcoCore.TcoMomentaryTask.On()"/> or <see cref="PlcDocu.TcoCore.TcoMomentaryTask.Off()"/> method call only when this property si '''TRUE'''.
        </summary>
    </docu>
~*)
PROPERTY Enabled : BOOL
GET
Enabled := _enabled;
END_GET
SET
_enabled := Enabled;

IF NOT _enabled THEN
    _state := FALSE;
    _setOnRequest := FALSE;
END_IF
END_SET
END_PROPERTY

(*~
    <docu>
        <summary>
            Gets identity of this instance.
            This value is assigned after download by calling the implicit method <c>FB_init()</c> and cannot be changed during runtime.
            This variable is used in the higher level applications.
        </summary>
    </docu>
~*)
PROPERTY Identity : ULINT
GET
Identity := _Identity;
END_GET
END_PROPERTY

PROPERTY IsOff : BOOL
GET
IsOff := NOT _state;
END_GET
END_PROPERTY

PROPERTY IsOn : BOOL
GET
IsOn := _state;
END_GET
END_PROPERTY

(*~
    <docu>
        <summary>
            Use to set the state of the '''TcoMomentaryTask''' to the value '''FALSE'''.
        </summary>
    </docu>
~*)
METHOD FINAL Off : BOOL
Off := FALSE;

//Check if Run method is called cyclically
IF THIS^.Context.StartCycleCount > _StartCycleCount + 1 THEN
    THIS^.Messenger.Programming('Run() method is not called cyclically.');
    RETURN;
END_IF

IF _state THEN
    THIS^._state := FALSE;
    OnFtrig();
    OnStateChange();
    Off := TRUE;
END_IF;
END_METHOD

(*~
    <docu>
        <summary>
            Use to set the state of the '''TcoMomentaryTask''' to the value '''TRUE'''.
        </summary>
    </docu>
~*)
METHOD FINAL On : BOOL
On := FALSE;

//Check if Run method is called cyclically
IF THIS^.Context.StartCycleCount > _StartCycleCount + 1 THEN
    THIS^.Messenger.Programming('Run() method is not called cyclically.');
    RETURN;
END_IF

IF _enabled THEN
    IF NOT _state THEN
        THIS^._state := TRUE;
        OnRtrig();
        OnStateChange();
        On := TRUE;
    END_IF;
ELSE
    THIS^.Messenger.Post('Toggletask cannot be set to TRUE as its Enabled property is FALSE.', eMessageCategory.Info);
END_IF
END_METHOD

(*~
    <docu>
        <summary>
            Executes when momentary task changes its state from '''TRUE''' to '''FALSE'''.
        </summary>
    </docu>
~*)
METHOD PROTECTED OnFtrig
END_METHOD

(*~
    <docu>
        <summary>
            Executes when momentary task changes its state from '''FALSE''' to '''TRUE'''.
        </summary>
    </docu>
~*)
METHOD PROTECTED OnRtrig
END_METHOD

(*~
    <docu>
        <summary>
            Executes when momentary task changes its state .
        </summary>
    </docu>
~*)
METHOD PROTECTED OnStateChange
END_METHOD

(*~
    <docu>
        <summary>
            This method needs to be called cyclically.
        </summary>
    </docu>
~*)
METHOD Run
VAR
    _serviceableParent : ITcoServiceable;
END_VAR
// Store the context start cycle. Used to detect if Run() method is called cyclically.
_StartCycleCount := THIS^.Context.StartCycleCount;

// Detects if parent is in serviceable state to enable manual invoke of the task from the HMI/SCADA system.
IF (THIS^.Parent <> 0) THEN
    _isServiceable := TRUE;

    IF (__QUERYINTERFACE(THIS^.Parent, _serviceableParent)) THEN
        IF (NOT _serviceableParent.IsService) THEN
            THIS^._setOnRequest := FALSE;
            _isServiceable := FALSE;
        END_IF
    END_IF
END_IF;

IF (THIS^._setOnRequest) THEN
    THIS^.On();
ELSE
    THIS^.Off();
END_IF;

IF _state THEN
    TaskOn();
ELSE
    TaskOff();
END_IF
END_METHOD

(*~
    <docu>
        <summary>
            Gets actual value of this instance.
        </summary>
    </docu>
~*)
PROPERTY State : BOOL
GET
State := _state;
END_GET
END_PROPERTY

(*~
    <docu>
        <summary>
            Executes when momentary task is in ```Off``` state .
        </summary>
    </docu>
~*)
METHOD PROTECTED TaskOff
END_METHOD

(*~
    <docu>
        <summary>
            Executes when momentary task is in  ```On``` state .
        </summary>
    </docu>
~*)
METHOD PROTECTED TaskOn
END_METHOD

END_FUNCTION_BLOCK

// ---- POUs/Prototypes/TcoSequencer/TcoSequence.TcPOU
FUNCTION_BLOCK TcoSequence EXTENDS TcoSequencerBase
VAR
    _openingClosingErrorMessenger : TcoMessenger(THIS^);
END_VAR

(*~
    <docu>
        <summary>
            In this `TcoSequence` implementation this method must be called after the last step of the sequence.
        </summary>
    </docu>
~*)
METHOD Close
i_Close();
END_METHOD

(*~
    <docu>
        <summary>
            <para>
                Completes the sequencer, and return the sequencer pointer to the first step in the seuqence.
                Method is typically called inside the last step of the sequence.
            </para>
        </summary>
    </docu>
~*)
METHOD PUBLIC FINAL CompleteSequence
i_CompleteSequence();
END_METHOD

(*~
    <docu>
        <summary>
            Completes the execution of the current step and moves the sequencer pointer to the next step in order of execution.
            The call returns `ITcoObjectRestorer` that allows to restore object upon step completition.
        </summary>
        <returns></returns>
    </docu>
~*)
METHOD PUBLIC FINAL CompleteStep : ITcoObjectRestorer
CompleteStep := i_CompleteStep();
END_METHOD

(*~
    <docu>
        <summary>
            Main method of the sequener. Custom code needs to be placed here. The sequencer is executed by call of **Instance.Run()** method.
            This method is abstract, and it must be overridden in derived block.
        </summary>
    </docu>
~*)
{attribute 'hide'}
{attribute 'obsolete' := 'Do not call this method explicitelly.'}
METHOD PROTECTED Main : BOOL
END_METHOD

(*~
    <docu>
        <summary>
            In this `TcoSequence` implementation this method must be called prior to first step call of the sequence.
        </summary>
    </docu>
~*)
METHOD Open
i_Open();
END_METHOD

(*~
    <docu>
        <summary>
            Terminates the currently executed step and set the sequencer's pointer to the step with Id that corresponds to ```inRequestedStepID``` parameter.
            When the order of the requested step is higher than the order of the currently finished step (the requested step is "after" the current one)
            the requested step is started in the same context cycle.
            When the order of the requested step is lower than the order of the currently finished step (the requested step is "before" the current one)
            the requested step is started in the next context cycle.
            If the requested step is not found even in the next context cycle, the sequencer enters error state ```StepWithRequestedIdDoesNotExists```.
            <para>
                See <see cref="TcoCore.eSequencerError"/> for detailed description.
            </para>
        </summary>
    </docu>
~*)
METHOD PUBLIC FINAL RequestStep : ITcoSequencer
VAR_INPUT
    (*~
        <docu>
            <summary>
                StepId of the step to be executed.
            </summary>
        </docu>
    ~*)
    inRequestedStepID : INT := MinStepID - 1;
END_VAR
VAR
    _message : STRING(254);
END_VAR
RequestStep := i_RequestStep(inRequestedStepID := inRequestedStepID);
END_METHOD

(*~
    <docu>
        <summary>
            <para>
                Ensures calling the Open(), Main() and Close() methods in the desired order.
                This method is final, so it cannot be overloaded. The **Instance.Run()** needs to be called cyclically inside the appropriate context.
            </para>
        </summary>
    </docu>
~*)
{attribute 'hide'}
{attribute 'obsolete' := 'Call of `Run` method does not have effect in this implementation.'}
METHOD PUBLIC FINAL Run
Messenger.Programming('Run method should not be called in this implementation of sequencer');
END_METHOD

METHOD PUBLIC Step : BOOL
VAR_INPUT
    (*~
    <docu>
        <summary>
            StepId of the current step.
            <remarks>
                <note type="important">
                    This number must be unique throughout the complete sequence.
                    It must be a constant or numerical literal and it must not change during the life-time of the sequencer.
                </note>
            </remarks>
        </summary>
    </docu>
~*)
    inStepID : INT;
    (*~
    <docu>
        <summary>
            If this value is false, step body is not executed and execution is moved to the next enabled step.
        </summary>
    </docu>
~*)
    inEnabled : BOOL;
    (*~
    <docu>
        <summary>
            Step description text.
        </summary>
    </docu>
~*)
    inStepDescription : STRING(254);
END_VAR
IF (_lastOpeningCycle <> Context.StartCycleCount) THEN
    _openingClosingErrorMessenger.Programming('Sequencer is not opened. You must call `Open` method before any step.');
END_IF

IF ((_lastOpeningCycle - _lastClosingCycle) > 1) THEN
    _openingClosingErrorMessenger.Programming('Sequencer is not closed. You must call `Close` method after last step call.');
END_IF

Step := i_Step(inStepID := inStepID, inEnabled := inEnabled, inStepDescription := inStepDescription);
END_METHOD

(*~
    <docu>
        <summary>
            Completes the actually running step, when the `inCondition` parameter is `TRUE`.
            Method is typically called inside a step as the transition method.
        </summary>
    </docu>
~*)
METHOD PUBLIC FINAL StepCompleteWhen
VAR_INPUT
    (*~
    <docu>
        <summary>
            The condition under which the step is completed.
        </summary>
    </docu>
~*)
    inCondition : BOOL;
END_VAR
i_StepCompleteWhen(inCondition := inCondition);
END_METHOD

END_FUNCTION_BLOCK

